//水冷泵测试
R_Test_watercooler_pump(CLK:=Test_watercooler_pump);
IF R_Test_watercooler_pump.Q AND (NOT Motor_work) AND (NOT cooler_motor_Test1)  THEN
    cooler_motor_Test:=TRUE;
	ELSIF R_Test_watercooler_pump.Q AND cooler_motor_Test1 THEN
    cooler_motor_Test:=FALSE;
END_IF
cooler_motor_Test1:=cooler_motor_Test;
//散热风扇测试
R_Test_cooler_fan(CLK:=Test_cooler_fan);
IF R_Test_cooler_fan.Q AND (NOT Motor_work) AND (NOT cooler_fan_Test1)  THEN
    cooler_fan_Test:=TRUE;
    ELSIF R_Test_cooler_fan.Q AND cooler_fan_Test1  THEN
    cooler_fan_Test:=FALSE;
END_IF
cooler_fan_Test1:=cooler_fan_Test;
//扫盘中速测试
R_Test_Sweep_Mspeed(CLK:=Test_Sweep_Mspeed);
IF R_Test_Sweep_Mspeed.Q AND (NOT Sweep_Mspeed_Test1)  THEN
    Sweep_Mspeed_Test:=TRUE;
    Sweep_Lspeed_Test:=FALSE;
ELSIF R_Test_Sweep_Mspeed.Q AND Sweep_Mspeed_Test1  THEN
    Sweep_Mspeed_Test:=FALSE;
END_IF
Sweep_Mspeed_Test1:=Sweep_Mspeed_Test;
//扫盘低速测试
R_Test_Sweep_Lspeed(CLK:=Test_Sweep_Lspeed);
IF R_Test_Sweep_Lspeed.Q AND (NOT Sweep_Lspeed_Test1)  THEN
    Sweep_Lspeed_Test:=TRUE;
    Sweep_Mspeed_Test:=FALSE;
ELSIF R_Test_Sweep_Lspeed.Q AND Sweep_Lspeed_Test1  THEN
    Sweep_Lspeed_Test:=FALSE;
END_IF
Sweep_Lspeed_Test1:=Sweep_Lspeed_Test;
//左扫旋转测试
R_Test_LSweep(CLK:=Test_LSweep);
IF R_Test_LSweep.Q AND (NOT LSweep_Test1)  THEN
    LSweep_Test:=TRUE;
    RSweep_Test:=FALSE;
    ASweep_Test:=FALSE;
ELSIF R_Test_LSweep.Q AND LSweep_Test1  THEN
    LSweep_Test:=FALSE;
END_IF
LSweep_Test1:=LSweep_Test;
//右扫旋转测试
R_Test_RSweep(CLK:=Test_RSweep);
IF R_Test_RSweep.Q AND (NOT RSweep_Test1) THEN
    RSweep_Test:=TRUE;
    LSweep_Test:=FALSE;
    ASweep_Test:=FALSE;
ELSIF R_Test_RSweep.Q AND RSweep_Test1  THEN
    RSweep_Test:=FALSE;
END_IF
RSweep_Test1:=RSweep_Test;
//全扫旋转测试
R_Test_ASweep(CLK:=Test_ASweep);
IF R_Test_ASweep.Q AND (NOT ASweep_Test1) THEN
    RSweep_Test:=FALSE;
    LSweep_Test:=FALSE;
    ASweep_Test:=TRUE;
ELSIF R_Test_ASweep.Q AND ASweep_Test1  THEN
    ASweep_Test:=FALSE;
END_IF
ASweep_Test1 :=ASweep_Test ;
//箱体升降测试
Box_Down_Test:=Test_Box_Down AND (NOT Test_Box_Up) AND (NOT DI_Rod_noDown);
Box_Up_Test:=Test_Box_Up AND (NOT Test_Box_Down);
//吸盘升降测试
Suction_Down_Test:=Test_Suction_Down AND (NOT Test_Suction_Up);
Suction_Up_Test:=Test_Suction_Up AND (NOT Test_Suction_Down);
//箱门开关测试
Boxdoor_close_Test:=Test_Door_Close AND (NOT Test_Door_Open);
Boxdoor_open_Test:=Test_Door_Open AND (NOT Test_Door_Close);
//左扫盘升降测试
LSweep_Up_Test:=Test_LSweep_Up AND (NOT Test_LSweep_Down) AND (NOT DI_Sweep_Down);
LSweep_Down_Test:=Test_LSweep_Down AND (NOT Test_LSweep_Up) AND (NOT DI_Sweep_Up);
//右扫盘升降测试
RSweep_Up_Test:=Test_RSweep_Up AND (NOT Test_RSweep_Down) AND (NOT DI_Sweep_Down);
RSweep_Down_Test:=Test_RSweep_Down AND (NOT Test_RSweep_Up) AND (NOT DI_Sweep_Up);
//左扫盘摆出测试
R_Test_LSweep_out(CLK:=Test_LSweep_out);
IF R_Test_LSweep_out.Q AND (NOT LSweep_out_Test1) THEN
    LSweep_out_Test:=TRUE;
ELSIF R_Test_LSweep_out.Q AND LSweep_out_Test1  THEN
    LSweep_out_Test:=FALSE;
END_IF
LSweep_out_Test1:=LSweep_out_Test;
//右扫盘摆出测试
R_Test_RSweep_out(CLK:=Test_RSweep_out);
IF R_Test_RSweep_out.Q AND (NOT RSweep_out_Test1) THEN
    RSweep_out_Test:=TRUE;
ELSIF R_Test_RSweep_out.Q AND RSweep_out_Test1  THEN
    RSweep_out_Test:=FALSE;
END_IF
RSweep_out_Test1:=RSweep_out_Test;
//左喷杆摆出测试
R_Test_Lrod_OUT(CLK:=Test_Lrod_OUT);
IF R_Test_Lrod_OUT.Q AND (NOT Lrod_OUT_Test1) THEN;
    Lrod_OUT_Test:=TRUE;
ELSIF R_Test_Lrod_OUT.Q AND Lrod_OUT_Test1 THEN;
    Lrod_OUT_Test:=FALSE;
END_IF
Lrod_OUT_Test1:=Lrod_OUT_Test;
//右喷杆摆出测试
R_Test_Rrod_OUT(CLK:=Test_Rrod_OUT);
IF R_Test_Rrod_OUT.Q AND (NOT Rrod_OUT_Test1) THEN;
    Rrod_OUT_Test:=TRUE;
ELSIF R_Test_Rrod_OUT.Q AND Rrod_OUT_Test1 THEN;
    Rrod_OUT_Test:=FALSE;
END_IF
Rrod_OUT_Test1 :=Rrod_OUT_Test;
//左喷杆喷水测试
R_Test_Lrod_water(CLK:=Test_Lrod_water);
IF R_Test_Lrod_water.Q AND (NOT Lrod_water_Test1) THEN
    Lrod_water_Test:=TRUE;
ELSIF R_Test_Lrod_water.Q AND Lrod_water_Test1 THEN
    Lrod_water_Test:=FALSE;
END_IF
Lrod_water_Test1:=Lrod_water_Test;
//右喷杆喷水测试
R_Test_Rrod_water(CLK:=Test_Rrod_water);
IF R_Test_Rrod_water.Q AND (NOT Rrod_water_Test1) THEN
    Rrod_water_Test:=TRUE;
ELSIF R_Test_Rrod_water.Q AND Rrod_water_Test1 THEN
    Rrod_water_Test:=FALSE;
END_IF
Rrod_water_Test1:=Rrod_water_Test;
//吸嘴喷杆喷水测试
R_Test_Suction_water(CLK:=Test_Suction_water);
IF R_Test_Suction_water.Q AND (NOT Suction_water_Test1) THEN
    Suction_water_Test:=TRUE;
ELSIF R_Test_Suction_water.Q AND Suction_water_Test1 THEN
    Suction_water_Test:=FALSE;
END_IF
Suction_water_Test1:=Suction_water_Test;
//高压冲洗测试
R_Test_Hpre_wash(CLK:=Test_Hpre_wash);
IF R_Test_Hpre_wash.Q AND (NOT Hpre_wash_Test1) THEN
    Hpre_wash_Test:=TRUE;
ELSIF R_Test_Hpre_wash.Q AND Hpre_wash_Test1 THEN
    Hpre_wash_Test:=FALSE;
END_IF
Hpre_wash_Test1:=Hpre_wash_Test;
//自洁测试
R_Test_selfclean(CLK:=Test_selfclean);
IF R_Test_selfclean.Q AND (NOT selfclean_water_Test1) THEN
    selfclean_water_Test:=TRUE;
END_IF
IF R_Test_selfclean.Q AND selfclean_water_Test1 THEN
    selfclean_water_Test:=FALSE;
END_IF
selfclean_water_Test1 :=selfclean_water_Test;
//高压水泵啮合测试
R_Test_Hpre_pump_gearin(CLK:=Test_Hpre_pump_gearin);
IF R_Test_Hpre_pump_gearin.Q AND (NOT Hpress_pump_gearin_Test1) THEN
    Hpress_pump_gearin_Test:=TRUE;
ELSIF (R_Test_Hpre_pump_gearin.Q AND Hpress_pump_gearin_Test1) OR T_pumpClutch.Q THEN
    Hpress_pump_gearin_Test:=FALSE;
END_IF
Hpress_pump_gearin_Test1 :=Hpress_pump_gearin_Test;
(*发动机工作时，水箱缺水时，延时10S高压水泵分离 *)
T_pumpClutch(IN:=Motor_work AND DI_cleanwater_LOW_ALM  AND Hpress_pump_gearin_Test ,PT:=T#10S);
//喷雾降尘泵测试
R_Test_fogpump(CLK:=Test_fogpump);
IF R_Test_fogpump.Q AND (NOT Fog_pump_Test1) THEN
    Fog_pump_Test:=TRUE;
ELSIF (R_Test_fogpump.Q AND Fog_pump_Test1) OR T_Fog_pump_Test.Q THEN
    Fog_pump_Test:=FALSE;
END_IF
Fog_pump_Test1 :=Fog_pump_Test;
(*发动机工作时，水箱缺水时，延时90S隔膜泵停止 *)
T_Fog_pump_Test(IN:=DI_cleanwater_LOW_ALM  AND Fog_pump_Test ,PT:=T#90S);
//污水泵测试
R_Test_wastewater_pump(CLK:=Test_wastewater_pump);
IF R_Test_wastewater_pump.Q AND (NOT Wastewater_pump_Test1) THEN
    Wastewater_pump_Test:=TRUE;
ELSIF R_Test_wastewater_pump.Q AND Wastewater_pump_Test1 THEN
    Wastewater_pump_Test:=FALSE;
END_IF
Wastewater_pump_Test1 :=Wastewater_pump_Test;
//污水泵球阀测试
R_Test_wastewater_valve(CLK:=Test_wastewater_valve);
IF R_Test_wastewater_valve.Q AND (NOT Wastewater_valve_Test1) THEN
    Wastewater_valve_Test:=TRUE;
ELSIF R_Test_wastewater_valve.Q AND Wastewater_valve_Test1 THEN
    Wastewater_valve_Test:=FALSE;
END_IF
Wastewater_valve_Test1 :=Wastewater_valve_Test;
//备用动力测试
R_Test_backup_power(CLK:=Test_backup_power);
IF R_Test_backup_power.Q AND (NOT Backup_power_Test1) THEN
    Backup_power_Test:=TRUE;
ELSIF (R_Test_backup_power.Q AND Backup_power_Test1) OR T_Backup_power_Test.Q THEN
    Backup_power_Test:=FALSE;
END_IF
Backup_power_Test1 :=Backup_power_Test;
(*备用动力打开90S后自动关闭 *)
T_Backup_power_Test(IN:=Backup_power_Test ,PT:=T#90S);
Backup_power_Test_warn:=Backup_power_Test AND (NOT DI_backup_power_open);

//点喷测试
Test_pointshoot_up := Pointshoot_up_Test AND NOT Pointshoot_down_Test;
Test_pointshoot_down := Pointshoot_down_Test AND NOT Pointshoot_up_Test; 
Test_pointshoot_left := Pointshoot_left_Test AND NOT Pointshoot_right_Test; 
Test_pointshoot_right := Pointshoot_right_Test AND NOT Pointshoot_left_Test;

END_PROGRAM

// Changsha_Xiangji_ARM_Cortex_A9_xilinx_zynq7000_linux/Application/CAN_COMM/prg_can0
PROGRAM prg_can0   //CAN0   与底盘和显示屏通信
VAR
	hCan0:CAA.HANDLE:=0;
    CanWriteData : ARRAY[0..7] OF BYTE;
    CanWriteMsgID:UDINT;
	CanReadData : ARRAY[0..7] OF BYTE;  
	CanReadMsgID:UDINT;
	bModifyTimeFlag :BOOL := FALSE;
	
	//通过CAN总线从底盘读到的信息
	can_data_ready:BOOL := FALSE;
	can_data_speed:BYTE := 0;
	can_data_soc:BYTE := 0;
	
	//通过CAN总线从显示屏读到的信息
	c00byte0bit0_both_wash_sweep:BOOL := FALSE;
	c00byte0bit1_left_wash_sweep:BOOL := FALSE;
	c00byte0bit2_right_wash_sweep:BOOL := FALSE;
	c00byte0bit3_both_sweep:BOOL := FALSE;
	c00byte0bit4_left_sweep:BOOL := FALSE;
	c00byte0bit5_right_sweep:BOOL := FALSE;
	c00byte0bit6_both_wash:BOOL := FALSE;
	c00byte0bit7_left_wash:BOOL := FALSE;
	
	c00byte1bit0_right_wash:BOOL := FALSE;
	c00byte1bit1_stop_sweep:BOOL := FALSE;
	c00byte1bit2_start_motor:BOOL := FALSE;
	c00byte1bit3_stop_motor:BOOL := FALSE;
	c00byte1bit4_speed_add:BOOL := FALSE;
	c00byte1bit5_speed_dec:BOOL := FALSE;
	c00byte1bit6_normal_speed:BOOL := FALSE;
	c00byte1bit7_high_speed:BOOL := FALSE;
	
	c00byte2bit0_garbage_close:BOOL := FALSE;
	c00byte2bit1_garbage_open:BOOL := FALSE;
	c00byte2bit2_garbage_up:BOOL := FALSE;
	c00byte2bit3_garbage_down:BOOL := FALSE;
	c00byte2bit4_fog_bump:BOOL := FALSE;
	c00byte2bit5_selfclean:BOOL := FALSE;
	c00byte2bit6_wastewater_pump:BOOL := FALSE;
	c00byte2bit7_res :BOOL := FALSE;
	
	c00byte3bit0_sweep_high:BOOL := FALSE;
	c00byte3bit1_sweep_middle:BOOL := FALSE;
	c00byte3bit2_sweep_low:BOOL := FALSE;
	c00byte3bit3_highpress_wash:BOOL := FALSE;
	c00byte3bit4_pointshoot_up:BOOL := FALSE;
	c00byte3bit5_pointshoot_down:BOOL := FALSE;
	c00byte3bit6_pointshoot_left:BOOL := FALSE;
	c00byte3bit7_pointshoot_right:BOOL := FALSE;

	c00byte4bit0_drain_start:BOOL := FALSE;
	c00byte4bit1_drain_auto:BOOL := FALSE;
	c00byte4bit2_drain_manual:BOOL := FALSE;
	c00byte4bit3_left_drain:BOOL := FALSE;
	c00byte4bit4_right_drain:BOOL := FALSE;
	c00byte4bit5_sub_drain:BOOL := FALSE;
	c00byte4bit6_selfclean_drain:BOOL := FALSE;
	c00byte4bit7_spout_drain:BOOL := FALSE;
	
	c00byte6bit0_func_test:BOOL := FALSE;
	c00byte6bit1_change_sweeper:BOOL := FALSE;
	c00byte6bit2_intelligent:BOOL := FALSE;
	c00byte6bit3_cleanly:BOOL := FALSE;
	c00byte6bit4_normal:BOOL := FALSE;
	c00byte6bit5_dirty:BOOL := FALSE;
	
	c01byte0bit3_test_watercooler_pump:BOOL := FALSE;
	c01byte0bit4_test_cooler_fan:BOOL := FALSE;
	
	c01byte1bit0_test_sweeper_middle:BOOL := FALSE;
	c01byte1bit1_test_sweeper_low:BOOL := FALSE;
	c01byte1bit2_test_left_sweeper:BOOL := FALSE;
	c01byte1bit3_test_right_sweeper:BOOL := FALSE;
	c01byte1bit4_test_both_sweeper:BOOL := FALSE;
	c01byte1bit5_test_box_down:BOOL := FALSE;
	c01byte1bit6_test_box_up:BOOL := FALSE;
	c01byte1bit7_test_sucker_down:BOOL := FALSE;
	
	c01byte2bit0_test_sucker_up:BOOL := FALSE;
	c01byte2bit1_test_box_open:BOOL := FALSE;
	c01byte2bit2_test_box_close:BOOL := FALSE;
	
	c01byte2bit6_test_left_sweeper_down:BOOL := FALSE;
	c01byte2bit7_test_left_sweeper_up:BOOL := FALSE;
	
	c01byte3bit0_test_right_sweeper_down:BOOL := FALSE;
	c01byte3bit1_test_right_sweeper_up:BOOL := FALSE;
	c01byte3bit2_test_left_sweeper_out:BOOL := FALSE;
	c01byte3bit3_test_right_sweeper_out:BOOL := FALSE;
	c01byte3bit4_test_left_shooter_out:BOOL := FALSE;
	c01byte3bit5_test_right_shooter_out:BOOL := FALSE;
	c01byte3bit6_test_left_shooter_water:BOOL := FALSE;
	c01byte3bit7_test_right_shooter_water:BOOL := FALSE;
	
	c01byte4bit0_test_sucker_water:BOOL := FALSE;
	c01byte4bit1_test_highpress_wash:BOOL := FALSE;
	c01byte4bit2_test_selfclean:BOOL := FALSE;
	c01byte4bit3_test_highpress_pump_gearin:BOOL := FALSE;
	c01byte4bit4_test_fogpump:BOOL := FALSE;
	c01byte4bit5_test_pointshoot_up:BOOL := FALSE;
    c01byte4bit6_test_pointshoot_down:BOOL := FALSE;
    c01byte4bit7_test_pointshoot_left:BOOL := FALSE;
	
	c01byte5bit0_test_pointshoot_right:BOOL := FALSE;
	c01byte5bit2_test_wastewater_pump:BOOL := FALSE;
	c01byte5bit3_test_wastewater_valve:BOOL := FALSE;
	
	c01byte6bit0_test_backup_power:BOOL := FALSE;
	
	c02byte45_speed_change :UINT := 0;
	c02byte67_sub_motor_min_speed:UINT := 0;
	
	c03byte01_normal_speed:UINT := 0;
	c03byte23_high_speed:UINT := 0;
	c03byte45_sweeper_speed:UINT := 0;
	
	c04byte01_highpress_pump_overspeed_warning:UINT := 0;
	c04byte23_highpress_pump_overspeed_stop:UINT := 0;
	c04byte45_sub_motor_max_speed:UINT := 0;
	c04byte67_sub_motor_idle_speed:UINT := 0;
	
	c05byte01_clean_low_speed:UINT := 0;
    c05byte23_clean_midlow_speed:UINT := 0;
    c05byte45_clean_midhigh_speed:UINT := 0;
    c05byte67_clean_high_speed:UINT := 0;
	
	c06byte01_normal_low_speed:UINT := 0;
    c06byte23_normal_midlow_speed:UINT := 0;
    c06byte45_normal_midhigh_speed:UINT := 0;
    c06byte67_normal_high_speed:UINT := 0;
	
	c07byte01_dirty_low_speed:UINT := 0;
    c07byte23_dirty_midlow_speed:UINT := 0;
    c07byte45_dirty_midhigh_speed:UINT := 0;
    c07byte67_dirty_high_speed:UINT := 0;
	
	//通过CAN总线发送到显示屏的信息
	s00byte0bit0_res:BOOL := FALSE;
	
	s00byte1bit0_res:BOOL := FALSE;
	s00byte1bit1_wastewater_full:BOOL := FALSE;
	s00byte1bit2_oil_filter_block:BOOL := FALSE;
	s00byte1bit3_oil_low:BOOL := FALSE;
	s00byte1bit4_res:BOOL := FALSE;
	s00byte1bit5_tank_no_water:BOOL := FALSE;
	s00byte1bit6_res:BOOL := FALSE;
	s00byte1bit7_back_error_stop:BOOL := FALSE;
	
	s00byte2bit0_wastewater_full_stop:BOOL := FALSE;
	s00byte2bit1_electronic_power_fault:BOOL := FALSE;
	s00byte2bit2_highpress_pump_overspeed_warning:BOOL := FALSE;
	s00byte2bit3_highpress_pump_overspeed_stop:BOOL := FALSE;
	s00byte2bit4_please_close_test:BOOL := FALSE;
	s00byte2bit5_being_back:BOOL := FALSE;
	s00byte2bit6_please_open_motor:BOOL := FALSE;
	s00byte2bit7_please_open_test:BOOL := FALSE;
	
	s00byte3bit0_air_press_low:BOOL := FALSE;
	s00byte3bit1_back_the_truck:BOOL := FALSE;
	s00byte3bit2_res:BOOL := FALSE;
	s00byte3bit3_highpress_pump_not_gearin:BOOL := FALSE;
	s00byte3bit4_water_valve_not_on:BOOL := FALSE;
	s00byte3bit5_highpress_blow_valve_not_on:BOOL := FALSE;
	s00byte3bit6_highpress_water_valve_not_on:BOOL := FALSE;
	s00byte3bit7_please_open_box_door:BOOL := FALSE;
	
	s00byte4bit0_pump_valve_not_no:BOOL := FALSE;
	s00byte4bit1_pump_press_fault:BOOL := FALSE;
	s00byte4bit2_fault_stop:BOOL := FALSE;
	s00byte4bit3_please_putdown_supporter:BOOL := FALSE;
	
	s00byte4bit6_chassis_can_fault:BOOL := FALSE;
	s00byte4bit7_motordriver_can_fault:BOOL :=FALSE;
	
	s00byte5bit0_sub_wastebox_error:BOOL := FALSE;
	s00byte5bit1_sub1_wastebox_full:BOOL := FALSE;
	s00byte5bit2_sub2_wastebox_full:BOOL := FALSE;
	s00byte5bit3_water_release_valve_not_close:BOOL := FALSE;
	s00byte5bit4_water_release_valve_not_copen:BOOL := FALSE;
	s00byte5bit5_backup_power_on:BOOL := FALSE;
	s00byte5bit6_power_low_20percent:BOOL := FALSE;
	s00byte5bit7_chassis_no_high_voltage:BOOL := FALSE;
	
	s00byte6bit0_cleanwater_LOW:BOOL := FALSE;
	s00byte6bit1_highpress_water_valve_on:BOOL := FALSE;
	s00byte6bit2_box_door_close:BOOL := FALSE;
	s00byte6bit3_highpress_blow_valve_on:BOOL := FALSE;
	s00byte6bit4_air_press_low:BOOL := FALSE;
	s00byte6bit5_wastewater_full:BOOL := FALSE;
	s00byte6bit6_supporter_nodown:BOOL := FALSE;
	s00byte6bit7_backup_power_open:BOOL := FALSE;
	
	s00byte7bit0_water_release_valve:BOOL := FALSE;
	s00byte7bit4_fog_pump_press_ok:BOOL := FALSE;
	s00byte7bit5_oil_level_low:BOOL := FALSE;
	s00byte7bit6_oil_filter_block:BOOL := FALSE;
	
	s01byte0bit0_power_on:BOOL := FALSE;
	s01byte0bit1_back_the_truck:BOOL := FALSE;
	s01byte0bit2_oil_release_valve:BOOL := FALSE;
	s01byte0bit3_cleanwater_low:BOOL := FALSE;
	s01byte0bit4_auxiliary1_warte_H:BOOL := FALSE;
	s01byte0bit5_auxiliary2_warte_H:BOOL := FALSE;
	s01byte0bit6_sweeper_up:BOOL := FALSE;
    s01byte0bit7_sweeper_down:BOOL := FALSE;
	
	s01byte1bit0_sweeper_out:BOOL := FALSE;
	s01byte1bit1_sweeper_return:BOOL := FALSE;
	
	s01byte3bit0_left_sweeper_down:BOOL := FALSE;
    s01byte3bit1_left_sweeper_up:BOOL := FALSE;
    s01byte3bit2_right_sweeper_down:BOOL := FALSE;
    s01byte3bit3_right_sweeper_up:BOOL := FALSE;
    s01byte3bit4_left_sweeper_out:BOOL := FALSE;
    s01byte3bit5_right_sweeper_out:BOOL := FALSE;
    s01byte3bit6_left_shooter_out:BOOL := FALSE;
    s01byte3bit7_right_shooter_out:BOOL := FALSE;

    s01byte4bit5_water_release_valve_open:BOOL := FALSE;
    s01byte4bit6_left_shooter_open:BOOL := FALSE;
    s01byte4bit7_right_shooter_open:BOOL := FALSE;
	
//	s01byte4bit4_oil_release_valve:BOOL := FALSE;
//	s01byte4bit5_sweeper_middle_speed:BOOL := FALSE;
//	s01byte4bit6_sweeper_low_speed:BOOL := FALSE;
//	s01byte4bit7_left_sweeper_back:BOOL := FALSE;
	
    s01byte5bit0_sucker_shooter_water:BOOL := FALSE;
    s01byte5bit1_fog_pump_open:BOOL := FALSE;
    s01byte5bit2_selfclean_shooter_water:BOOL := FALSE;
    s01byte5bit3_high_sub_shooter_water:BOOL := FALSE;
    s01byte5bit4_Spump_open:BOOL := FALSE;
    s01byte5bit5_engine_en:BOOL := FALSE;
    s01byte5bit6_watercooler_pump_open:BOOL := FALSE;
    s01byte5bit7_cooler_fan_open:BOOL := FALSE;
	
    s01byte6bit0_backup_power_open:BOOL := FALSE;
    s01byte6bit1wastewater_valve_open:BOOL := FALSE;
    s01byte6bit2_wastewater_pump_open:BOOL := FALSE;
    s01byte6bit3_oil_release_valve_open:BOOL := FALSE;
    s01byte6bit4_sweep_middle_open:BOOL := FALSE;
    s01byte6bit5_sweep_low_open:BOOL := FALSE;
    s01byte6bit6_right_sweep_open:BOOL := FALSE;
    s01byte6bit7_left_both_sweep_open:BOOL := FALSE;
	
    s01byte7bit0_right_both_sweep_open:BOOL := FALSE;
    s01byte7bit1_box_down:BOOL := FALSE;
    s01byte7bit2_box_up:BOOL := FALSE;
    s01byte7bit3_sucker_down:BOOL := FALSE;
    s01byte7bit4_sucker_up:BOOL := FALSE;
    s01byte7bit5_box_open:BOOL := FALSE;
    s01byte7bit6_box_close:BOOL := FALSE;
	
	s02byte0bit67_right_shooter_out:BYTE := 0;
	
	s02byte1bit01_left_shooter_out:BYTE := 0;
	s02byte1bit23_waterpump_gearin:BYTE := 0;
	s02byte1bit45_left_shooter_valve_open:BYTE := 0;
	s02byte1bit67_right_shooter_valve_open:BYTE := 0;
	
	s02byte2bit01_sucker_shooter_valve_open:BYTE := 0;
	s02byte2bit23_selfclean_shooter_valve_open:BYTE := 0;
	s02byte2bit45_high_sub_shooter_valve_open:BYTE := 0;
	s02byte2bit67_water_release_valve:BYTE := 0;
	
	s02byte3bit01_oil_release_valve:BYTE := 0;
	s02byte3bit23_sweeper_middle_speed:BYTE := 0;
	s02byte3bit45_sweeper_low_speed:BYTE := 0;
	s02byte3bit67_left_sweeper_back:BYTE := 0;
	
	s02byte4bit01_left_sweeper_down:BYTE := 0;
	s02byte4bit23_right_sweeper_back:BYTE := 0;
	s02byte4bit45_right_sweeper_down:BYTE := 0;
	s02byte4bit67_left_all_sweep:BYTE := 0;
	
	s02byte5bit01_right_sweep:BYTE := 0;
	s02byte5bit23_res:BYTE := 0;
	
	s02byte6bit01_right_all_sweep:BYTE := 0;
	s02byte6bit23_box_down:BYTE := 0;
	s02byte6bit45_box_up:BYTE := 0;
	s02byte6bit67_sucker_up:BYTE := 0;
	
	s02byte7bit01_sucker_down:BYTE := 0;
	s02byte7bit23_boxdoor_close:BYTE := 0;
	s02byte7bit45_boxdoor_open:BYTE := 0;
	s02byte7bit67_cleanwater_pump:BYTE := 0;
	
	s03byte0bit01_res:BYTE := 0;
	s03byte0bit23_water_coller_motor:BYTE := 0;
	s03byte0bit45_cooler_fan:BYTE := 0;
	s03byte0bit67_lowpress_pump:BYTE := 0;
	
	s03byte3bit0_all_wash_sweep:BOOL := FALSE;
	s03byte3bit1_left_wash_sweep:BOOL := FALSE;
	s03byte3bit2_right_wash_sweep:BOOL := FALSE;
	s03byte3bit3_all_sweep:BOOL := FALSE;
	s03byte3bit4_left_sweep:BOOL := FALSE;
	s03byte3bit5_right_sweep:BOOL := FALSE;
	s03byte3bit6_all_wash:BOOL := FALSE;
	s03byte3bit7_left_wash:BOOL := FALSE;
	
	s03byte4bit0_right_wash:BOOL := FALSE;
	s03byte4bit1_stop_sweep:BOOL := FALSE;
	s03byte4bit2_fog_pump:BOOL := FALSE;
	s03byte4bit3_selfclean:BOOL := FALSE;
	s03byte4bit4_boxdoor_close:BOOL := FALSE;
	s03byte4bit5_boxdoor_open:BOOL := FALSE;
	s03byte4bit6_box_up:BOOL := FALSE;
	s03byte4bit7_box_down:BOOL := FALSE;
	
	s03byte5bit0_motor_start:BOOL := FALSE;
	s03byte5bit1_motor_stop:BOOL := FALSE;
	s03byte5bit4_normal_speed:BOOL := FALSE;
	s03byte5bit5_high_speed:BOOL := FALSE;
	s03byte5bit6_sweeper_high_speed:BOOL := FALSE;
	s03byte5bit7_sweeper_middle_spped:BOOL := FALSE;
	
	s03byte6bit0_sweeper_low_speed:BOOL := FALSE;
	s03byte6bit1_highpress_wash:BOOL := FALSE;
	s03byte6bit2_drain_start:BOOL := FALSE;
	s03byte6bit3_drain_auto:BOOL := FALSE;
	s03byte6bit4_drain_manual:BOOL := FALSE;
	s03byte6bit5_drain_left_shooter:BOOL := FALSE;
	s03byte6bit6_drain_right_shooter:BOOL := FALSE;
	s03byte6bit7_sub_drain:BOOL := FALSE;
	
	s03byte7bit0_drain_selfclean:BOOL := FALSE;
	s03byte7bit1_change_sweeper:BOOL := FALSE;
	s03byte7bit2_func_test:BOOL := FALSE;
	s03byte7bit3_intelligent:BOOL := FALSE;
	s03byte7bit4_cleanly:BOOL := FALSE;
	s03byte7bit5_normal:BOOL := FALSE;
	s03byte7bit6_dirty:BOOL := FALSE;
	s03byte7bit7_wastewater_pump:BOOL := FALSE;
	
	s04byte0bit0_point_shoot_up:BOOL := FALSE;
	s04byte0bit1_point_shoot_down:BOOL := FALSE;
	s04byte0bit2_point_shoot_left:BOOL := FALSE;
	s04byte0bit3_point_shoot_right:BOOL := FALSE;
	s04byte0bit4_sucker_shooter_drain:BOOL := FALSE;
	
	s04byte1bit3_test_cooler_motor:BOOL := FALSE;
	s04byte1bit4_test_cooler_fan:BOOL := FALSE;
	s04byte1bit5_test_sweeper_middle:BOOL := FALSE;
	s04byte1bit6_test_sweeper_low:BOOL := FALSE;
	s04byte1bit7_test_left_sweep:BOOL := FALSE;
	
	s04byte2bit0_test_right_sweep:BOOL := FALSE;
	s04byte2bit1_test_all_sweep:BOOL := FALSE;
	s04byte2bit2_test_box_down:BOOL := FALSE;
	s04byte2bit3_test_box_up:BOOL := FALSE;
	s04byte2bit4_test_sucker_down:BOOL := FALSE;
	s04byte2bit5_test_sucker_up:BOOL := FALSE;
	s04byte2bit6_test_boxdoor_open:BOOL := FALSE;
	s04byte2bit7_test_boxdoor_close:BOOL := FALSE;
	
	s04byte3bit0_test_left_sweeper_down:BOOL := FALSE;
	s04byte3bit1_test_left_sweeper_up:BOOL := FALSE;
	s04byte3bit2_test_right_sweeper_down:BOOL := FALSE;
	s04byte3bit3_test_right_sweeper_up:BOOL := FALSE;
	s04byte3bit4_test_left_shooter_out:BOOL := FALSE;
	s04byte3bit5_test_right_shooter_out:BOOL := FALSE;
	s04byte3bit6_test_left_shooter_water:BOOL := FALSE;
	s04byte3bit7_test_right_shooter_water:BOOL := FALSE;
	
	s04byte4bit0_test_sucker_water:BOOL := FALSE;
	s04byte4bit1_test_highpress_wash:BOOL := FALSE;
	s04byte4bit2_test_selfclean:BOOL := FALSE;
	s04byte4bit3_test_highpress_pump_gearin:BOOL := FALSE;
	s04byte4bit4_test_fog_pump:BOOL := FALSE;
	s04byte4bit5_test_left_sweeper_out:BOOL := FALSE;
	s04byte4bit6_test_right_sweeper_out:BOOL := FALSE;
	s04byte4bit7_test_wastewater_pump:BOOL := FALSE;
	
	s04byte5bit0_test_wastewater_valve:BOOL := FALSE;
	s04byte5bit1_test_backup_power:BOOL := FALSE;
	s04byte5bit6_motor_starting:BOOL := FALSE;
	s04byte5bit7_system_running:BOOL := FALSE;
	
	s05byte45_speed_change_value:UINT := 0;
	s05byte67_sub_motor_min_speed:UINT := 0;
	
	s06byte01_normal_speed:UINT := 0;
	s06byte23_high_speed:UINT := 0;
	s06byte45_sweeper_speed:UINT := 0;
	
	s07byte01_highpress_pump_high_speed:UINT := 0;
	s07byte23_highpress_pump_high_speed_stop:UINT := 0;
	s07byte45_sub_motor_max_speed:UINT := 0;
	s07byte67_sub_motor_idle_speed:UINT := 0;
	
	s08byte01_real_torque:UINT := 0;
	s08byte23_real_speed:UINT := 0;
	s08byte45_bus_voltage:UINT := 0;
	s08byte67_phase_current:UINT := 0;
	
	s09byte01_max_dirve_torque:UINT := 0;
	s09byte23_max_brake_torque:UINT := 0;
	s09byte4_temp_controller:BYTE := 0;
	s09byte5_temp_motor:BYTE := 0;
	s09byte67_motor_max_speed:UINT := 0;
	
	s10byte0bit23_direction_cw:BYTE := 0;
	s10byte0bit45_motor_mode:BYTE := 0;
	s10byte0bit67_motor_stat:BYTE := 0;
	
	s10byte1bit01_bus_low_voltage:BYTE := 0;
	s10byte1bit23_bus_high_voltage:BYTE := 0;
	s10byte1bit45_ctrller_high_temp:BYTE := 0;
	s10byte1bit67_motor_high_temp:BYTE := 0;
	
	s10byte2bit01_igbt_fault:BYTE := 0;
	s10byte2bit23_overspeed:BYTE := 0;
	s10byte2bit45_comm_error:BYTE := 0;
	s10byte2bit67_short:BYTE := 0;
	
	s10byte3bit01_motor_overload:BYTE := 0;
	s10byte3bit23_selfcheck_fault:BYTE := 0;
	s10byte3bit45_low_voltage:BYTE := 0;
	s10byte3bit67_sensor_fault:BYTE := 0;
	
	s11byte0_chassis_power_percent:BYTE := 0;
	s11byte1_res :BYTE := 0;
	s11byte23_speed_set_value:UINT := 0;
	s11byte45_version:UINT := 0;
	
    //电机
	
	hReceiver1:CAA.HANDLE;
	hReceiver2:CAA.HANDLE;
	hReceiver3:CAA.HANDLE;
	
	//显示屏 0x0c00 074f ~ 0x0c07 074f
	hRecver_screen:CAA.HANDLE;
	
	tmp_byte:BYTE;
	tmp_uint:UINT;
	Err:CAA.ERROR;
	
	hMsg : CAA.HANDLE;
	nReceived : CAA.COUNT;
	nAvailable: CAA.COUNT;
	ReadErr   : CAA.ERROR;
	MsgID     : CL2I.COBID;	
	pRxData :POINTER TO CL2I.DATA;
	//电机CAN通信标志位
	nReceived1 : CAA.COUNT;
	
	can_stat : DINT := 0;
	
	n: INT := 0;
	m: INT := 0;
END_VAR

CASE can_stat OF
	0:   //init can port0 and port1
		hCan0 := cl2.DriverOpenH(usiNetId:=0,uiBaudRate:=250,xSupport29Bits:=TRUE,ctMessages:=100,peError:=ADR(Err));	 //CAN1
		IF hCan0 > 0 THEN
			can_stat := 10;
		END_IF
	
	10: //create receiver for data
		//接收驱动器信息1: ID:0x0C112AEE,  
	  	hReceiver1 := CL2.CreateMaskReceiver(hDriver := hCan0,
			cobIdValue := 16#0C112AEE, //cobID value
			cobIdMask := 16#FFFFFFFF, //cobID mask ==> all bits of value are relevant									
			xRTRValue := FALSE, //no RTR messages
			xRTRMask := FALSE, //activate RTR filter ==> xRTRValue will be checked
			x29BitIdValue := TRUE, //29 bit CAN messages
			x29BitIdMask := TRUE, //activate 29 bit filter ==> x29BitIdValue will be checked
			xTransmitValue := FALSE, //only receive messages, no transmit message loopback
			xTransmitMask := FALSE, //activate transmit mask filter ==> xTransmitValue will be checked
			xAlwaysNewest := FALSE, //FALSE := receiver with queue; TRUE: only newest message
			eEvent := CB.EVENT.NO_EVENT,  //no receive event
			xEnableSyncWindow := FALSE, //not implemented
			peError := ADR(Err) //optional pointer to error
			);
		//接收驱动器信息2: ID:0x0C122AEE	
	  	hReceiver2 := CL2.CreateMaskReceiver(hDriver := hCan0,
			cobIdValue := 16#0C122AEE, //cobID value
			cobIdMask := 16#FFFFFFFF, //cobID mask ==> all bits of value are relevant									
			xRTRValue := FALSE, //no RTR messages
			xRTRMask := FALSE, //activate RTR filter ==> xRTRValue will be checked
			x29BitIdValue := TRUE, //29 bit CAN messages
			x29BitIdMask := TRUE, //activate 29 bit filter ==> x29BitIdValue will be checked
			xTransmitValue := FALSE, //only receive messages, no transmit message loopback
			xTransmitMask := FALSE, //activate transmit mask filter ==> xTransmitValue will be checked
			xAlwaysNewest := FALSE, //FALSE := receiver with queue; TRUE: only newest message
			eEvent := CB.EVENT.NO_EVENT, //no receive event
			xEnableSyncWindow := FALSE, //not implemented
			peError := ADR(Err) //optional pointer to error
			);	
		
		//接收驱动器信息3: ID:0x0C132AEE
		hReceiver3 := CL2.CreateMaskReceiver(hDriver := hCan0,
			cobIdValue := 16#0C132AEE, //cobID value
			cobIdMask := 16#FFFFFFFF, //cobID mask ==> all bits of value are relevant									
			xRTRValue := FALSE, //no RTR messages
			xRTRMask := FALSE, //activate RTR filter ==> xRTRValue will be checked
			x29BitIdValue := TRUE, //no 29 bit CAN messages
			x29BitIdMask := TRUE, //activate 29 bit filter ==> x29BitIdValue will be checked
			xTransmitValue := FALSE, //only receive messages, no transmit message loopback
			xTransmitMask := FALSE, //activate transmit mask filter ==> xTransmitValue will be checked
			xAlwaysNewest := FALSE, //FALSE := receiver with queue; TRUE: only newest message
			eEvent := CB.EVENT.NO_EVENT, //no receive event
			xEnableSyncWindow := FALSE, //not implemented
			peError := ADR(Err) //optional pointer to error
		);
				//创建接收显示屏信息的接收器: ID:0x0cxx074f
		hRecver_screen := CL2.CreateMaskReceiver(hDriver := hCan0,
			cobIdValue := 16#0C00074F, //cobID value  
			cobIdMask := 16#FFF8FFFF, //cobID mask	0c00074f,0c01074f,0c02074f,0c03074f,							
			xRTRValue := FALSE, //no RTR messages
			xRTRMask := FALSE, //activate RTR filter ==> xRTRValue will be checked
			x29BitIdValue := TRUE, //no 29 bit CAN messages
			x29BitIdMask := TRUE, //activate 29 bit filter ==> x29BitIdValue will be checked
			xTransmitValue := FALSE, //only receive messages, no transmit message loopback
			xTransmitMask := FALSE, //activate transmit mask filter ==> xTransmitValue will be checked
			xAlwaysNewest := FALSE, //FALSE := receiver with queue; TRUE: only newest message
			eEvent := CB.EVENT.NO_EVENT, //no receive event
			xEnableSyncWindow := FALSE, //not implemented
			peError := ADR(Err) //optional pointer to error
		);
		
		IF (hReceiver1 <> 0 AND hReceiver2 <> 0 AND hReceiver3 <> 0 AND hRecver_screen <> 0) THEN
			 can_stat := 20;
		ELSE
			RETURN;
		END_IF
	20:  //receive data
		//接收驱动器信息1: ID:0x0C112AEE,  
		nReceived1 := cl2.GetMsgCount(hReceiverId :=hReceiver1, peError := ADR(ReadErr));
		m:=m+1;
		WHILE nReceived1 > 0 DO
			m:=0;
			hMsg := cl2.Read(hReceiverId :=hReceiver1,pctMsgLeft:=ADR(nAvailable),peError:=ADR(ReadErr));
			pRxData := cl2.GetMessageDataPointer(hMessage:= hMsg,peError:=ADR(ReadErr));	
			get_buf_0C112AEE(pRxData);
			cl2.FreeMessage(hMsg);
	        nReceived1 := cl2.GetMsgCount(hReceiverId :=hReceiver1, peError := ADR(ReadErr));
		END_WHILE


		//接收驱动器信息2: ID:0x0C122AEE
		nReceived1 := cl2.GetMsgCount(hReceiverId :=hReceiver2, peError := ADR(ReadErr));
		WHILE nReceived1 > 0 DO
			hMsg := cl2.Read(hReceiverId :=hReceiver2,pctMsgLeft:=ADR(nAvailable),peError:=ADR(ReadErr));
			pRxData := cl2.GetMessageDataPointer(hMessage:= hMsg,peError:=ADR(ReadErr));	
			get_buf_0C122AEE(pRxData);
			cl2.FreeMessage(hMsg);
			nReceived1 := cl2.GetMsgCount(hReceiverId :=hReceiver2, peError := ADR(ReadErr));
		END_WHILE

		//接收驱动器信息3: ID:0x0C132AEE
		nReceived1 := cl2.GetMsgCount(hReceiverId :=hReceiver3, peError := ADR(ReadErr));
		WHILE nReceived1 > 0 DO
			hMsg := cl2.Read(hReceiverId :=hReceiver3,pctMsgLeft:=ADR(nAvailable),peError:=ADR(ReadErr));
			pRxData := cl2.GetMessageDataPointer(hMessage:= hMsg,peError:=ADR(ReadErr));	
			get_buf_0C132AEE(pRxData);
			cl2.FreeMessage(hMsg);	
			nReceived1 := cl2.GetMsgCount(hReceiverId :=hReceiver3, peError := ADR(ReadErr));
		END_WHILE
        
		
       //接收显示屏信息: ID:0x0cXX074f
		nReceived := cl2.GetMsgCount(hReceiverId :=hRecver_screen, peError := ADR(ReadErr));
		n:=n+1;
		WHILE nReceived > 0 DO
			n:=0;
			hMsg := cl2.Read(hReceiverId :=hRecver_screen,pctMsgLeft:=ADR(nAvailable),peError:=ADR(ReadErr));
			pRxData := cl2.GetMessageDataPointer(hMessage:= hMsg,peError:=ADR(ReadErr));	
			MsgID := cl2.GetMessageId(hMessage := hMsg, peError := ADR(ReadErr));
			proc_screen_data(MsgID := MsgID, pRxData := pRxData);
			cl2.FreeMessage(hMsg);		
			nReceived := cl2.GetMsgCount(hReceiverId :=hRecver_screen, peError := ADR(ReadErr));	
		END_WHILE
		(*
		IF nReceived <> 0 THEN
			hMsg := cl2.Read(hReceiverId :=hRecver_screen,pctMsgLeft:=ADR(nAvailable),peError:=ADR(ReadErr));
			pRxData := cl2.GetMessageDataPointer(hMessage:= hMsg,peError:=ADR(ReadErr));	
			MsgID := cl2.GetMessageId(hMessage := hMsg, peError := ADR(ReadErr));
			proc_screen_data(MsgID := MsgID, pRxData := pRxData);
			cl2.FreeMessage(hMsg);
		END_IF	
		nReceived := cl2.GetMsgCount(hReceiverId :=hRecver_screen, peError := ADR(ReadErr));
		IF nReceived <> 0 THEN
			hMsg := cl2.Read(hReceiverId :=hRecver_screen,pctMsgLeft:=ADR(nAvailable),peError:=ADR(ReadErr));
			pRxData := cl2.GetMessageDataPointer(hMessage:= hMsg,peError:=ADR(ReadErr));	
			MsgID := cl2.GetMessageId(hMessage := hMsg, peError := ADR(ReadErr));
			proc_screen_data(MsgID := MsgID, pRxData := pRxData);
			cl2.FreeMessage(hMsg);
		END_IF	
		*)
		//与电机CAN通讯失败
        T_Motor_CAN_fault(IN:=m>100,PT:=T#1S);
		//与屏通讯失败
        T_Screen_CAN_fault(IN:=n>100,PT:=T#1S);		
		can_stat := 30;
		
		
	30: //send data 
		//send data to motor
		set_buf_0801EE2A();
		CAN_Send_MSG(hCan0, 16#0801EE2A, 8, CanWriteData);
		
		//send data to screen
		// 12帧数据一起发送，以后可以根据需要调整发送间隔
		set_buf_18004f07();
		CAN_Send_MSG(hCan0, 16#18004F07, 8, CanWriteData);	
		
		set_buf_18014f07();
		CAN_Send_MSG(hCan0, 16#18014F07, 8, CanWriteData);	
			
		set_buf_18024f07();
		CAN_Send_MSG(hCan0, 16#18024F07, 8, CanWriteData);	
		
		set_buf_18034f07();
		CAN_Send_MSG(hCan0, 16#18034F07, 8, CanWriteData);	
	
		set_buf_18044f07();
		CAN_Send_MSG(hCan0, 16#18044F07, 8, CanWriteData);			
		
		set_buf_18054f07();
		CAN_Send_MSG(hCan0, 16#18054F07, 8, CanWriteData);			
		
		set_buf_18064f07();
		CAN_Send_MSG(hCan0, 16#18064F07, 8, CanWriteData);	
		
		set_buf_18074f07();
		CAN_Send_MSG(hCan0, 16#18074F07, 8, CanWriteData);	
		
		set_buf_18084f07();
		CAN_Send_MSG(hCan0, 16#18084F07, 8, CanWriteData);	
		
		set_buf_18094f07();
		CAN_Send_MSG(hCan0, 16#18094F07, 8, CanWriteData);	

		set_buf_18104f07();
		CAN_Send_MSG(hCan0, 16#18104F07, 8, CanWriteData);	

		set_buf_18114f07();
		CAN_Send_MSG(hCan0, 16#18114F07, 8, CanWriteData);	
		
		set_buf_18124f07();
		CAN_Send_MSG(hCan0, 16#18124F07, 8, CanWriteData);

		set_buf_18134f07();
		CAN_Send_MSG(hCan0, 16#18134F07, 8, CanWriteData);

		set_buf_18144f07();
		CAN_Send_MSG(hCan0, 16#18144F07, 8, CanWriteData);
	
		can_stat := 20;
	
	
	100:   //error
END_CASE

METHOD set_buf_18004f07 : bool
VAR_INPUT
END_VAR

VAR
	tmp_byte : BYTE := 0;
	tmp_uint: UINT := 0;
END_VAR
tmp_byte := 0;
CanWriteData[0] := tmp_byte;

tmp_byte := 0;
tmp_byte.0 := FALSE;
tmp_byte.1 := Wastewater_full_Fault;//污水满故障
tmp_byte.2 := T_DI_oil_filter_block.Q;//回油过滤堵塞
tmp_byte.3 := T_DI_oil_level_low.Q;//液压油位低故障
tmp_byte.4 := s00byte1bit4_res;
tmp_byte.5 := T_DI_cleanwater_LOW.Q;//水箱缺水故障
tmp_byte.6 := s00byte1bit6_res;
tmp_byte.7 := DI_Rcar_fault;//倒车故障停机
CanWriteData[1] := tmp_byte;

tmp_byte := 0;
tmp_byte.0 := Wastewater_full_Fault1;//污水满故障停机
tmp_byte.1 := NOT DI_power_on;//电源故障
tmp_byte.2 := T_Pumpspeed_H.Q;//高压水泵超速报警
tmp_byte.3 := T_Pumpspeed_HH.Q;//高压水泵超速停止
tmp_byte.4 := TEST_ALM;//请关闭测试
tmp_byte.5 := RCAR_ALM;//正在倒车中提示
tmp_byte.6 := Motor_Work_ALM;//请先启动电机提示
tmp_byte.7 := Func_test_HMI;//测试打开
CanWriteData[2] := tmp_byte;

tmp_byte := 0;
tmp_byte.0 := T_DI_air_press_low.Q;//气路系统压力低
tmp_byte.1 := T_DI_Rcar.Q;//倒车
tmp_byte.2 := s00byte3bit2_res;
tmp_byte.3 := DO_Hpre_pump_noWork;//高压水泵未啮合
tmp_byte.4 := T_Chassis_SOC_LOW.Q;//底盘电量低停机
tmp_byte.5 := DI_Hpre_valve_noOpen;//高压吹净球阀未打开
tmp_byte.6 := DI_Totvalve_noOpen;//高压水路球阀未打开
tmp_byte.7 := DO_Box_Up_arm;//请先打开箱门
CanWriteData[3] := tmp_byte;

tmp_byte := 0;
tmp_byte.0 := fog_Spump_arm;//隔膜泵球阀未打开
tmp_byte.1 := T_fog_pump_press_noOk.Q;//隔膜泵压力不正常
tmp_byte.2 := Fault_STOP;//故障停机
tmp_byte.3 := DO_Box_Down_arm;//请先放下撑杆
tmp_byte.4 := T_DI_wastewater_full.Q;//主污水箱水满
tmp_byte.5 := Backup_power_Test_warn;//请先打开备用动力开关
tmp_byte.6 := T_Chassis_CAN_fault.Q;//底盘CAN通讯故障
tmp_byte.7 := T_Motor_CAN_fault.Q;//与电机CAN通讯故障
CanWriteData[4] := tmp_byte;

tmp_byte := 0;
tmp_byte.0 := T_auxiliary_warte_dif.Q;//辅污水箱水位不一致
tmp_byte.1 := T_DI_auxiliary1_warte_H.Q;//辅1污水箱水满
tmp_byte.2 := T_DI_auxiliary2_warte_H.Q;//辅2污水箱水满
tmp_byte.3 := T_water_overflow_noClose.Q;//水路卸荷阀未关闭故障
tmp_byte.4 := T_water_overflow_noOpen.Q;//水路卸荷阀未打开故障
tmp_byte.5 := DI_backup_power_open;//备用动力打开提示
tmp_byte.6 := Chassis_SOC_LOW;//底盘电量低压20%提示
tmp_byte.7 := High_voltage_noReady;//底盘未上高压提示
CanWriteData[5] := tmp_byte;

tmp_byte := 0;
tmp_byte.0 := (DI_cleanwater_LOW<3000);
tmp_byte.1 := DI_Totvalve_Open;
tmp_byte.2 := DI_box_door_close;
tmp_byte.3 := DI_Hpre_valve_open;
tmp_byte.4 := DI_air_press_low;
tmp_byte.5 := DI_wastewater_full;
tmp_byte.6 := DI_Rod_noDown;
tmp_byte.7 := DI_backup_power_open;
CanWriteData[6] := tmp_byte;

tmp_byte := 0;
tmp_byte.0 := DI_water_overflow;
tmp_byte.1 := FALSE;
tmp_byte.2 := FALSE;
tmp_byte.3 := FALSE;
tmp_byte.4 := DI_fog_pump_press_ok;
tmp_byte.5 := DI_oil_level_low;
tmp_byte.6 := DI_oil_filter_block;
tmp_byte.7 := FALSE;
CanWriteData[7] := tmp_byte;

set_buf_18004f07 := TRUE;
END_METHOD

METHOD set_buf_18074f07 : bool
VAR_INPUT
END_VAR

VAR
	tmp_byte : BYTE := 0;
	tmp_uint: UINT := 0;
END_VAR
tmp_byte := ANY_TO_BYTE(S_Pumpspeed_arm MOD 256);
CanWriteData[0] := tmp_byte;

tmp_byte := ANY_TO_BYTE(S_Pumpspeed_arm/256);
CanWriteData[1] := tmp_byte;

tmp_byte := ANY_TO_BYTE(S_Pumpspeed_stop MOD 256);
CanWriteData[2] := tmp_byte;

tmp_byte := ANY_TO_BYTE(S_Pumpspeed_stop/256);
CanWriteData[3] := tmp_byte;

tmp_byte := ANY_TO_BYTE(S_MAX_Speed MOD 256);
CanWriteData[4] := tmp_byte;

tmp_byte := ANY_TO_BYTE(S_MAX_Speed/256);
CanWriteData[5] := tmp_byte;

tmp_byte := ANY_TO_BYTE(S_Idle_Speed MOD 256);
CanWriteData[6] := tmp_byte;

tmp_byte := ANY_TO_BYTE(S_Idle_Speed/256);
CanWriteData[7] := tmp_byte;

set_buf_18074f07 := TRUE;
END_METHOD

METHOD get_buf_0c00074f : bool
VAR_INPUT
	pRxData :POINTER TO CL2I.DATA;
END_VAR

VAR
	tmp_byte : BYTE := 0;

END_VAR
tmp_byte := pRxData^[0];
HMI_Awashsweep := tmp_byte.0;
HMI_Lwashsweep := tmp_byte.1;
HMI_Rwashsweep:= tmp_byte.2;
HMI_Asweeproad := tmp_byte.3;
HMI_Lsweeproad := tmp_byte.4;
HMI_Rsweeproad := tmp_byte.5;
HMI_Acleanwash := tmp_byte.6;
HMI_Lcleanwash := tmp_byte.7;

tmp_byte := pRxData^[1];
HMI_Rcleanwash:= tmp_byte.0;
HMI_stop_sweep:= tmp_byte.1;
HMI_start_motor := tmp_byte.2;
HMI_stop_motor := tmp_byte.3;
HMI_Inc_Speed:= tmp_byte.4;
HMI_Dec_Speed:= tmp_byte.5;
HMI_Standard_speed := tmp_byte.6;
HMI_Strong_speed := tmp_byte.7;

tmp_byte := pRxData^[2];
HMI_Door_Close := tmp_byte.0;
HMI_Door_Open := tmp_byte.1;
HMI_Box_Up:= tmp_byte.2;
HMI_Box_Down:= tmp_byte.3;
HMI_fog_Spump:= tmp_byte.4;
HMI_selfclean := tmp_byte.5;
HMI_wastewater_pump := tmp_byte.6;
c00byte2bit7_res := tmp_byte.7;

tmp_byte := pRxData^[3];
HMI_Sweep_Hspd:= tmp_byte.0;
HMI_Sweep_Mspd:= tmp_byte.1;
HMI_Sweep_Lspd:= tmp_byte.2;
HMI_Hpre_wash := tmp_byte.3;
HMI_pointshoot_up := tmp_byte.4;
HMI_pointshoot_down := tmp_byte.5;
HMI_pointshoot_left := tmp_byte.6;
HMI_pointshoot_right := tmp_byte.7;

tmp_byte := pRxData^[4];
HMI_drain_start := tmp_byte.0;
HMI_drain_auto := tmp_byte.1;
HMI_drain_manual := tmp_byte.2;
HMI_Lrod_drain := tmp_byte.3;
HMI_Rrod_drain := tmp_byte.4;
HMI_Hpressure_drain := tmp_byte.5;
HMI_selfclean_drain := tmp_byte.6;
HMI_Suction_drain := tmp_byte.7;

tmp_byte := pRxData^[6];
HMI_func_test := tmp_byte.0;
HMI_replace_Sweep:= tmp_byte.1;
HMI_intelligent := tmp_byte.2;
HMI_cleanly := tmp_byte.3;
HMI_normal := tmp_byte.4;
HMI_dirty := tmp_byte.5;
	
get_buf_0c00074f := TRUE;
END_METHOD

METHOD proc_screen_data : bool
VAR_INPUT
	MsgID     : CL2I.COBID;	
	pRxData :POINTER TO CL2I.DATA;
END_VAR
CASE MsgID OF
	16#0C00074F:
		get_buf_0c00074f(pRxData);
	16#0C01074F:
		get_buf_0c01074f(pRxData);
	16#0C02074F:
		get_buf_0c02074f(pRxData);
	16#0C03074F:
		get_buf_0c03074f(pRxData);	
	16#0C04074F:
		get_buf_0c04074f(pRxData);	
	16#0C05074F:
		get_buf_0c05074f(pRxData);
	16#0C06074F:
		get_buf_0c06074f(pRxData);
	16#0C07074F:
		get_buf_0c07074f(pRxData);	
END_CASE
END_METHOD

METHOD set_buf_18104f07 : bool
VAR_INPUT
END_VAR

VAR
	tmp_byte : BYTE := 0;
	tmp_uint: UINT := 0;
END_VAR

tmp_byte := 0;
tmp_byte := tmp_byte + 0*1;
tmp_byte := tmp_byte + Motor_direction_cw*4;
tmp_byte := tmp_byte + Motor_mode*16;
tmp_byte := tmp_byte + Motor_stat*64;
CanWriteData[0] := tmp_byte;

tmp_byte := 0;
tmp_byte := tmp_byte + Motor_bus_low_voltage*1;
tmp_byte := tmp_byte + Motor_bus_high_voltage*4;
tmp_byte := tmp_byte + MOtor_ctrller_high_temp*16;
tmp_byte := tmp_byte + Motor_high_temp*64;
CanWriteData[1] := tmp_byte;

tmp_byte := 0;
tmp_byte := tmp_byte + Motor_igbt_fault*1;
tmp_byte := tmp_byte + Motor_overspeed*4;
tmp_byte := tmp_byte + Motor_comm_error*16;
tmp_byte := tmp_byte + Motor_short*64;
CanWriteData[2] := tmp_byte;

tmp_byte := 0;
tmp_byte := tmp_byte + Motor_overload*1;
tmp_byte := tmp_byte + Motor_selfcheck_fault*4;
tmp_byte := tmp_byte + Motor_low_voltage*16;
tmp_byte := tmp_byte + Motor_sensor_fault*64;
CanWriteData[3] := tmp_byte;
	

set_buf_18104f07 := TRUE;
END_METHOD

METHOD set_buf_0801EE2A : BOOL
VAR_INPUT
END_VAR

VAR
	tmp_byte : BYTE := 0;
	tmp_uint: UINT := 0;
END_VAR
tmp_byte := ANY_TO_BYTE(16#19 MOD 256);
CanWriteData[0] := tmp_byte;
tmp_byte := ANY_TO_BYTE(0/256);
CanWriteData[1] := tmp_byte;

tmp_byte := ANY_TO_BYTE(0 MOD 256);
CanWriteData[2] := tmp_byte;
tmp_byte := ANY_TO_BYTE(SETspeed_PID MOD 256);
CanWriteData[3] := tmp_byte;

tmp_byte := ANY_TO_BYTE(SETspeed_PID/256);
CanWriteData[4] := tmp_byte;
tmp_byte := ANY_TO_BYTE(0/256);
CanWriteData[5] := tmp_byte;

tmp_byte := ANY_TO_BYTE(0 MOD 256);
CanWriteData[6] := tmp_byte;
tmp_byte := ANY_TO_BYTE(0/256);
CanWriteData[7] := tmp_byte;

set_buf_0801EE2A := TRUE;
END_METHOD

METHOD get_buf_0C112AEE : BOOL
VAR_INPUT
	pRxData :POINTER TO CL2I.DATA;
END_VAR

VAR

END_VAR
Motor_real_torque_HMI := 256*ANY_TO_UINT(pRxData^[1]) + ANY_TO_UINT(pRxData^[0]);
Motor_real_speed_HMI :=  256*ANY_TO_UINT(pRxData^[3]) + ANY_TO_UINT(pRxData^[2]);
Motor_bus_voltage_HMI :=  256*ANY_TO_UINT(pRxData^[5]) + ANY_TO_UINT(pRxData^[4]);
Motor_phase_current_HMI :=  256*ANY_TO_UINT(pRxData^[7]) + ANY_TO_UINT(pRxData^[6]);

get_buf_0C112AEE := TRUE;
END_METHOD

METHOD set_buf_18114f07 : bool
VAR_INPUT
END_VAR

VAR
	tmp_byte : BYTE := 0;
	tmp_uint: UINT := 0;
END_VAR
//tmp_byte := ANY_TO_BYTE(s09byte23_max_brake_torque/256);
//CanWriteData[3] := tmp_byte;

CanWriteData[0] := Chassis_Soc;//底盘电量
//CanWriteData[1] := s11byte0_chassis_power_percent;

tmp_byte := ANY_TO_BYTE(SETspeed_PID MOD 256);
CanWriteData[2] := tmp_byte;//设定电机转速
tmp_byte := ANY_TO_BYTE(SETspeed_PID/256);
CanWriteData[3] := tmp_byte;

tmp_byte := ANY_TO_BYTE(16#201 MOD 256);
CanWriteData[4] := tmp_byte;//程序版本
tmp_byte := ANY_TO_BYTE(16#201/256);
CanWriteData[5] := tmp_byte;

tmp_byte :=ANY_TO_BYTE(Chassis_speed MOD 256);// ANY_TO_BYTE(Chassis_speed MOD 256);
CanWriteData[6] := tmp_byte;//底盘车速
tmp_byte :=ANY_TO_BYTE(Chassis_speed/256); //ANY_TO_BYTE(Chassis_speed/256);
CanWriteData[7] := tmp_byte;

set_buf_18114f07 := TRUE;
END_METHOD

METHOD set_buf_18044f07 : bool
VAR_INPUT
END_VAR

VAR
	tmp_byte : BYTE := 0;
	tmp_uint: UINT := 0;
END_VAR

tmp_byte := 0;
tmp_byte.0 := Pointshoot_up_HMI;
tmp_byte.1 := Pointshoot_down_HMI;
tmp_byte.2 := Pointshoot_left_HMI;
tmp_byte.3 := Pointshoot_right_HMI;
tmp_byte.4 := Suction_drain_HMI;
tmp_byte.5 := FALSE;
tmp_byte.6 := FALSE;
tmp_byte.7 := FALSE;
CanWriteData[0] := tmp_byte;

tmp_byte := 0;
tmp_byte.0 := FALSE;
tmp_byte.1 := FALSE;
tmp_byte.2 := FALSE;
tmp_byte.3 := cooler_motor_Test;
tmp_byte.4 := cooler_fan_Test;
tmp_byte.5 := Sweep_Mspeed_Test;
tmp_byte.6 := Sweep_Lspeed_Test;
tmp_byte.7 := LSweep_Test;
CanWriteData[1] := tmp_byte;
	
tmp_byte := 0;
tmp_byte.0 := RSweep_Test;
tmp_byte.1 := ASweep_Test;
tmp_byte.2 := Box_Down_Test;
tmp_byte.3 := Box_Up_Test;
tmp_byte.4 := Suction_Down_Test;
tmp_byte.5 := Suction_Up_Test;
tmp_byte.6 := Boxdoor_open_Test;
tmp_byte.7 := Boxdoor_close_Test;
CanWriteData[2] := tmp_byte;

	
tmp_byte := 0;
tmp_byte.0 := LSweep_Down_Test;
tmp_byte.1 := LSweep_Up_Test;
tmp_byte.2 := RSweep_Down_Test;
tmp_byte.3 := RSweep_Up_Test;
tmp_byte.4 := Lrod_OUT_Test;
tmp_byte.5 := Rrod_OUT_Test;
tmp_byte.6 := Lrod_water_Test;
tmp_byte.7 := Rrod_water_Test;
CanWriteData[3] := tmp_byte;
	
tmp_byte := 0;
tmp_byte.0 := Suction_water_Test;
tmp_byte.1 := Hpre_wash_Test;
tmp_byte.2 := selfclean_water_Test;
tmp_byte.3 := Hpress_pump_gearin_Test;
tmp_byte.4 := Fog_pump_Test;
tmp_byte.5 := LSweep_out_Test;
tmp_byte.6 := RSweep_out_Test;
tmp_byte.7 := Wastewater_pump_Test;
CanWriteData[4] := tmp_byte;

tmp_byte := 0;
tmp_byte.0 := Wastewater_valve_Test;
tmp_byte.1 := Backup_power_Test;
tmp_byte.2 := Pointshoot_up_Test;
tmp_byte.3 := Pointshoot_down_Test;
tmp_byte.4 := Pointshoot_left_Test;
tmp_byte.5 := Pointshoot_right_Test;
tmp_byte.6 := Motor_Work;
tmp_byte.7 := SYS_work;
CanWriteData[5] := tmp_byte;

set_buf_18044f07 := TRUE;
END_METHOD

METHOD set_buf_18024f07 : bool
VAR_INPUT
END_VAR

VAR
	tmp_byte : BYTE := 0;
	tmp_uint: UINT := 0;
	
END_VAR
tmp_byte := 0;
tmp_byte.0:=DO_Lsweep_down_short;
tmp_byte.1:=DO_Lsweep_down_open;
tmp_byte.2:=DO_Lsweep_up_short;
tmp_byte.3:=DO_Lsweep_up_open;
tmp_byte.4:=DO_Rsweep_down_short;
tmp_byte.5:=DO_Rsweep_down_open;
tmp_byte.6:=DO_Rsweep_up_short;
tmp_byte.7:=DO_Rsweep_up_open;
CanWriteData[0] := tmp_byte;

tmp_byte := 0;
tmp_byte.0:=DO_Lsweep_out_short;
tmp_byte.1:=DO_Lsweep_out_open;
tmp_byte.2:=DO_Rsweep_out_short;
tmp_byte.3:=DO_Rsweep_out_open;
tmp_byte.4:=DO_Lrod_out_short;
tmp_byte.5:=DO_Lrod_out_open;
tmp_byte.6:=DO_Rrod_out_short;
tmp_byte.7:=DO_Rrod_out_open;
CanWriteData[1] := tmp_byte;

tmp_byte := 0;
tmp_byte.0:=DO_pointshoot_up_short;
tmp_byte.1:=DO_pointshoot_up_open;
tmp_byte.2:=DO_pointshoot_Down_short;
tmp_byte.3:=DO_pointshoot_Down_open;
tmp_byte.4:=DO_pointshoot_left_short;
tmp_byte.5:=DO_pointshoot_left_open;
tmp_byte.6:=DO_pointshoot_right_short;
tmp_byte.7:=DO_pointshoot_right_open;
CanWriteData[2] := tmp_byte;

tmp_byte := 0;
//tmp_byte.0:=;
//tmp_byte.1:=;
tmp_byte.2:=DO_water_overflow_short;
tmp_byte.3:=DO_water_overflow_open;
tmp_byte.4:=DO_Lrod_water_short;
tmp_byte.5:=DO_Lrod_water_open;
tmp_byte.6:=DO_Rrod_water_short;
tmp_byte.7:=DO_Rrod_water_open;
CanWriteData[3] := tmp_byte;

tmp_byte := 0;
tmp_byte.0:=DO_Suction_water_short;
tmp_byte.1:=DO_Suction_water_open;
tmp_byte.2:=DO_Hpressure_water_short;
tmp_byte.3:=DO_Hpressure_water_open;
tmp_byte.4:=DO_selfclean_water_short;
tmp_byte.5:=DO_selfclean_water_open;
tmp_byte.6:=DO_Hpre_pump_short;
tmp_byte.7:=DO_Hpre_pump_open;
CanWriteData[4] := tmp_byte;

tmp_byte := 0;
tmp_byte.0:=DO_fog_Spump_short;
tmp_byte.1:=DO_fog_Spump_open;
tmp_byte.2:=DO_Motor_en_short;
tmp_byte.3:=DO_Motor_en_open;
tmp_byte.4:=DO_watercooler_pump_short;
tmp_byte.5:=DO_watercooler_pump_open;
tmp_byte.6:=DO_cooler_fan_short;
tmp_byte.7:=DO_cooler_fan_open;
CanWriteData[5] := tmp_byte;

tmp_byte := 0;
tmp_byte.0:=DO_backup_power_short;
tmp_byte.1:=DO_backup_power_open;
//tmp_byte.2:=;
//tmp_byte.3:=;
//tmp_byte.4:=;
//tmp_byte.5:=;
//tmp_byte.6:=;
//tmp_byte.7:=;
CanWriteData[6] := tmp_byte;

tmp_byte := 0;
(*
tmp_byte.0:=;
tmp_byte.1:=;
tmp_byte.2:=;
tmp_byte.3:=;
tmp_byte.4:=;
tmp_byte.5:=;
tmp_byte.6:=;
tmp_byte.7:=;
*)
CanWriteData[7] := tmp_byte;
	
set_buf_18024f07 := TRUE;
END_METHOD

METHOD set_buf_18014f07 : bool
VAR_INPUT
END_VAR

VAR
	tmp_byte : BYTE := 0;
	tmp_uint: UINT := 0;
END_VAR
tmp_byte := 0;
tmp_byte.0 := DI_power_on;
tmp_byte.1 := DI_Rcar;
tmp_byte.2 := DI_oil_release_valve;
tmp_byte.3 := FALSE;
tmp_byte.4 := DI_auxiliary1_warte_H;
tmp_byte.5 := DI_auxiliary2_warte_H;
tmp_byte.6 := DI_Sweep_Up;
tmp_byte.7 := DI_Sweep_Down;
CanWriteData[0] := tmp_byte;

tmp_byte := 0;
tmp_byte.0 := DI_sweep_out;//s01byte1bit0_box_down;
tmp_byte.1 := DI_sweep_return;//s01byte1bit1_box_up;
tmp_byte.2 := FALSE;//s01byte1bit2_sucker_down;
tmp_byte.3 := FALSE;//s01byte1bit3_sucker_up;
tmp_byte.4 := FALSE;//s01byte1bit4_boxdoor_close;
tmp_byte.5 := FALSE;//s01byte1bit5_boxdoor_open;
tmp_byte.6 := FALSE;//s01byte1bit6_shooter_out;
tmp_byte.7 := FALSE;//s01byte1bit7_shooter_return;
CanWriteData[1] := tmp_byte;

tmp_byte := 0;
tmp_byte.0 :=  FALSE;//s01byte2bit0_right_sweeper_up;
tmp_byte.1 :=  FALSE;//s01byte2bit1_right_sweeper_down;
tmp_byte.2 :=  FALSE;//s01byte2bit2_cleanwater_high;
tmp_byte.3 := FALSE;// s01byte2bit3_alterable_box_low;
tmp_byte.4 := FALSE;// s01byte2bit4_res;
tmp_byte.5 := FALSE;
tmp_byte.6 := FALSE;
tmp_byte.7 := FALSE;
CanWriteData[2] := tmp_byte;

tmp_byte := 0;
tmp_byte.0 := DO_Lsweep_down;
tmp_byte.1 := DO_Lsweep_up;
tmp_byte.2 := DO_Rsweep_down;
tmp_byte.3 := DO_Rsweep_up;
tmp_byte.4 := DO_Lsweep_out;
tmp_byte.5 := DO_Rsweep_out;
tmp_byte.6 := DO_Lrod_out;
tmp_byte.7 := DO_Rrod_out;
CanWriteData[3] := tmp_byte;

tmp_byte := 0;
tmp_byte.0 :=  DO_pointshoot_up;
tmp_byte.1 :=  DO_pointshoot_down;
tmp_byte.2 :=  DO_pointshoot_left;
tmp_byte.3 :=  DO_pointshoot_right;
tmp_byte.4 :=  FALSE;//s01byte4bit4_oil_release_valve;//
tmp_byte.5 := DO_water_overflow;
tmp_byte.6 := DO_Lrod_water;
tmp_byte.7 := DO_Rrod_water;
CanWriteData[4] := tmp_byte;


tmp_byte := 0;
tmp_byte.0 := DO_Suction_water;
tmp_byte.1 := DO_Hpressure_water;
tmp_byte.2 := DO_selfclean_water;
tmp_byte.3 := DO_Hpre_pump;
tmp_byte.4 := DO_fog_Spump;
tmp_byte.5 := DO_Motor_en;
tmp_byte.6 := DO_watercooler_pump;
tmp_byte.7 := DO_cooler_fan;
CanWriteData[5] := tmp_byte;


tmp_byte := 0;
tmp_byte.0 := DO_backup_power;
tmp_byte.1 := DO_wastewater_valve;
tmp_byte.2 := DO_wastewater_pump;
tmp_byte.3 := DO_oil_release_valve;
tmp_byte.4 := DO_Sweep_Mspeed;
tmp_byte.5 := DO_Sweep_Lspeed;
tmp_byte.6 := DO_RSweep;
tmp_byte.7 := DO_LASweep;
CanWriteData[6] := tmp_byte;

tmp_byte := 0;
tmp_byte.0 := DO_RASweep;
tmp_byte.1 := DO_Box_Down;
tmp_byte.2 := DO_Box_Up;
tmp_byte.3 := DO_Suction_Down;
tmp_byte.4 := DO_Suction_Up;
tmp_byte.5 := DO_Door_Open;
tmp_byte.6 := DO_Door_Close;
tmp_byte.7 := FALSE;
CanWriteData[7] := tmp_byte;

set_buf_18014f07 := TRUE;
END_METHOD

METHOD get_buf_0c02074f : bool
VAR_INPUT
	pRxData :POINTER TO CL2I.DATA;
END_VAR

VAR
	tmp_byte : BYTE := 0;
	tmp_uint: UINT := 0;
END_VAR

Re_IncDec_Speed:= 256*ANY_TO_UINT(pRxData^[5]) + ANY_TO_UINT(pRxData^[4]);
Re_motor_min_speed := 256*ANY_TO_UINT(pRxData^[7]) + ANY_TO_UINT(pRxData^[6]);

get_buf_0c02074f := TRUE;
END_METHOD

METHOD get_buf_0C132AEE : BOOL
VAR_INPUT
	pRxData :POINTER TO CL2I.DATA;
END_VAR

VAR
	tmp_byte : BYTE := 0;
	tmp_uint: UINT := 0;
END_VAR
Motor_direction_cw := ANY_TO_BYTE(pRxData^[0]/4)MOD 4;
Motor_mode := ANY_TO_BYTE(pRxData^[0]/16) MOD 4;
Motor_stat := ANY_TO_BYTE(pRxData^[0]/64)MOD 4;

Motor_bus_low_voltage := ANY_TO_BYTE(pRxData^[1]/1)MOD 4;
Motor_bus_high_voltage := ANY_TO_BYTE(pRxData^[1]/4)MOD 4;
MOtor_ctrller_high_temp := ANY_TO_BYTE(pRxData^[1]/16)MOD 4;
Motor_high_temp := ANY_TO_BYTE(pRxData^[1]/64)MOD 4;

Motor_igbt_fault := ANY_TO_BYTE(pRxData^[2]/1)MOD 4;
Motor_overspeed := ANY_TO_BYTE(pRxData^[2]/4)MOD 4;
Motor_comm_error := ANY_TO_BYTE(pRxData^[2]/16)MOD 4;
Motor_short := ANY_TO_BYTE(pRxData^[2]/64)MOD 4;

Motor_overload := ANY_TO_BYTE(pRxData^[3]/1)MOD 4;
Motor_selfcheck_fault := ANY_TO_BYTE(pRxData^[3]/4)MOD 4;
Motor_low_voltage := ANY_TO_BYTE(pRxData^[3]/16)MOD 4;
Motor_sensor_fault := ANY_TO_BYTE(pRxData^[3]/64)MOD 4;


get_buf_0C132AEE := TRUE;
END_METHOD

METHOD get_buf_0c05074f : bool
VAR_INPUT
	pRxData :POINTER TO CL2I.DATA;
END_VAR

Re_clean_low_speed := 256*ANY_TO_UINT(pRxData^[1]) + ANY_TO_UINT(pRxData^[0]);
Re_clean_midlow_speed := 256*ANY_TO_UINT(pRxData^[3]) + ANY_TO_UINT(pRxData^[2]);
Re_clean_midhigh_speed := 256*ANY_TO_UINT(pRxData^[5]) + ANY_TO_UINT(pRxData^[4]);
Re_clean_high_speed := 256*ANY_TO_UINT(pRxData^[7]) + ANY_TO_UINT(pRxData^[6]);

get_buf_0c05074f := TRUE;
END_METHOD

METHOD get_buf_0c04074f : bool
VAR_INPUT
	pRxData :POINTER TO CL2I.DATA;
END_VAR

Re_Pumpspeed_arm:= 256*ANY_TO_UINT(pRxData^[1]) + ANY_TO_UINT(pRxData^[0]);
Re_Pumpspeed_stop:= 256*ANY_TO_UINT(pRxData^[3]) + ANY_TO_UINT(pRxData^[2]);
Re_MAX_Speed:= 256*ANY_TO_UINT(pRxData^[5]) + ANY_TO_UINT(pRxData^[4]);
Re_Idle_Speed := 256*ANY_TO_UINT(pRxData^[7]) + ANY_TO_UINT(pRxData^[6]);

get_buf_0c04074f := TRUE;
END_METHOD

METHOD set_buf_18054f07 : bool
VAR_INPUT
END_VAR

VAR
	tmp_byte : BYTE := 0;
	tmp_uint: UINT := 0;
END_VAR
tmp_byte := ANY_TO_BYTE(S_IncDec_Speed MOD 256);
CanWriteData[4] := tmp_byte;

tmp_byte := ANY_TO_BYTE(S_IncDec_Speed/256);
CanWriteData[5] := tmp_byte;

tmp_byte := ANY_TO_BYTE(S_min_speed MOD 256);
CanWriteData[6] := tmp_byte;

tmp_byte := ANY_TO_BYTE(S_min_speed/256);
CanWriteData[7] := tmp_byte;

set_buf_18054f07 := TRUE;
END_METHOD

METHOD get_buf_0c01074f : bool
VAR_INPUT
	pRxData :POINTER TO CL2I.DATA;
END_VAR

VAR
	tmp_byte : BYTE := 0;
	tmp_uint: UINT := 0;
END_VAR
tmp_byte := pRxData^[0];
Test_watercooler_pump := tmp_byte.3;
Test_cooler_fan := tmp_byte.4;

tmp_byte := pRxData^[1];
Test_Sweep_Mspeed:= tmp_byte.0;
Test_Sweep_Lspeed:= tmp_byte.1;
Test_LSweep:= tmp_byte.2;
Test_RSweep:= tmp_byte.3;
Test_ASweep:= tmp_byte.4;
Test_Box_Down:= tmp_byte.5;
Test_Box_Up:= tmp_byte.6;
Test_Suction_Down:= tmp_byte.7;

tmp_byte := pRxData^[2];
Test_Suction_Up:= tmp_byte.0;
Test_Door_Open:= tmp_byte.1;
Test_Door_Close:= tmp_byte.2;
Test_LSweep_Down:= tmp_byte.6;
Test_LSweep_Up:= tmp_byte.7;

tmp_byte := pRxData^[3];
Test_RSweep_Down:= tmp_byte.0;
Test_RSweep_Up:= tmp_byte.1;
Test_LSweep_out := tmp_byte.2;
Test_RSweep_out := tmp_byte.3;
Test_Lrod_OUT:= tmp_byte.4;
Test_Rrod_OUT:= tmp_byte.5;
Test_Lrod_water:= tmp_byte.6;
Test_Rrod_water:= tmp_byte.7;

tmp_byte := pRxData^[4];
Test_Suction_water:= tmp_byte.0;
Test_Hpre_wash:= tmp_byte.1;
Test_selfclean:= tmp_byte.2;
Test_Hpre_pump_gearin := tmp_byte.3;
Test_fogpump := tmp_byte.4;
Test_pointshoot_up := tmp_byte.5;
Test_pointshoot_down := tmp_byte.6;
Test_pointshoot_left := tmp_byte.7;

tmp_byte := pRxData^[5];
Test_pointshoot_right := tmp_byte.0;
Test_wastewater_pump := tmp_byte.2;
Test_wastewater_valve := tmp_byte.3;

tmp_byte := pRxData^[6];
Test_backup_power := tmp_byte.0;

get_buf_0c01074f := TRUE;
END_METHOD

METHOD get_buf_0C122AEE : BOOL
VAR_INPUT
	pRxData :POINTER TO CL2I.DATA;
END_VAR

VAR
	tmp_byte : BYTE := 0;
	tmp_uint: UINT := 0;
END_VAR
Motor_max_dirve_torque_HMI := 256*ANY_TO_UINT(pRxData^[1]) + ANY_TO_UINT(pRxData^[0]);
Motor_max_brake_torque_HMI :=  256*ANY_TO_UINT(pRxData^[3]) + ANY_TO_UINT(pRxData^[2]);
Motor_temp_controller_HMI  := ANY_TO_BYTE(pRxData^[4]);
Motor_temp_HMI  := ANY_TO_BYTE(pRxData^[5]);

Motor_max_speed_HMI :=  256*ANY_TO_UINT(pRxData^[7]) + ANY_TO_UINT(pRxData^[6]);

get_buf_0C122AEE := TRUE;
END_METHOD

METHOD set_buf_18124f07 : BOOL
VAR_INPUT
END_VAR

VAR
	tmp_byte : BYTE := 0;
	tmp_uint: UINT := 0;
END_VAR

tmp_byte := ANY_TO_BYTE(S_clean_low_speed MOD 256);
CanWriteData[0] := tmp_byte;
tmp_byte := ANY_TO_BYTE(S_clean_low_speed/256);
CanWriteData[1] := tmp_byte;

tmp_byte := ANY_TO_BYTE(S_clean_midlow_speed MOD 256);
CanWriteData[2] := tmp_byte;
tmp_byte := ANY_TO_BYTE(S_clean_midlow_speed/256);
CanWriteData[3] := tmp_byte;

tmp_byte := ANY_TO_BYTE(S_clean_midhigh_speed MOD 256);
CanWriteData[4] := tmp_byte;
tmp_byte := ANY_TO_BYTE(S_clean_midhigh_speed/256);
CanWriteData[5] := tmp_byte;

tmp_byte := ANY_TO_BYTE(S_clean_high_speed MOD 256);
CanWriteData[6] := tmp_byte;
tmp_byte := ANY_TO_BYTE(S_clean_high_speed/256);
CanWriteData[7] := tmp_byte;

set_buf_18124f07 := TRUE;
END_METHOD

METHOD set_buf_18084f07 : bool
VAR_INPUT
END_VAR

VAR
	tmp_byte : BYTE := 0;
	tmp_uint: UINT := 0;
END_VAR
tmp_byte := ANY_TO_BYTE(Motor_real_torque_HMI MOD 256);
CanWriteData[0] := tmp_byte;

tmp_byte := ANY_TO_BYTE(Motor_real_torque_HMI/256);
CanWriteData[1] := tmp_byte;

IF Motor_real_speed_HMI<5 THEN
   Motor_real_speed_HMI:=0;
   ELSE
	Motor_real_speed_HMI:=Motor_real_speed_HMI;   
END_IF
                 
tmp_byte := ANY_TO_BYTE(Motor_real_speed_HMI MOD 256);
CanWriteData[2] := tmp_byte;

tmp_byte := ANY_TO_BYTE(Motor_real_speed_HMI/256);
CanWriteData[3] := tmp_byte;

tmp_byte := ANY_TO_BYTE(Motor_bus_voltage_HMI MOD 256);
CanWriteData[4] := tmp_byte;

tmp_byte := ANY_TO_BYTE(Motor_bus_voltage_HMI/256);
CanWriteData[5] := tmp_byte;

tmp_byte := ANY_TO_BYTE(Motor_phase_current_HMI MOD 256);
CanWriteData[6] := tmp_byte;

tmp_byte := ANY_TO_BYTE(Motor_phase_current_HMI/256);
CanWriteData[7] := tmp_byte;


set_buf_18084f07 := TRUE;
END_METHOD

METHOD set_buf_18064f07 : bool
VAR_INPUT
END_VAR


VAR
	tmp_byte : BYTE := 0;
	tmp_uint: UINT := 0;
END_VAR

tmp_byte := ANY_TO_BYTE(S_Standard_Speed MOD 256);
CanWriteData[0] := tmp_byte;

tmp_byte := ANY_TO_BYTE(S_Standard_Speed/256);
CanWriteData[1] := tmp_byte;

tmp_byte := ANY_TO_BYTE(S_Strong_Speed MOD 256);
CanWriteData[2] := tmp_byte;

tmp_byte := ANY_TO_BYTE(S_Strong_Speed/256);
CanWriteData[3] := tmp_byte;

tmp_byte := ANY_TO_BYTE(S_Sweep_Speed MOD 256);
CanWriteData[4] := tmp_byte;

tmp_byte := ANY_TO_BYTE(S_Sweep_Speed/256);
CanWriteData[5] := tmp_byte;

set_buf_18064f07 := TRUE;
END_METHOD

METHOD set_buf_18144f07 : BOOL
VAR_INPUT
END_VAR

VAR
	tmp_byte : BYTE := 0;
	tmp_uint: UINT := 0;
END_VAR

tmp_byte := ANY_TO_BYTE(S_dirty_low_speed MOD 256);
CanWriteData[0] := tmp_byte;
tmp_byte := ANY_TO_BYTE(S_dirty_low_speed/256);
CanWriteData[1] := tmp_byte;

tmp_byte := ANY_TO_BYTE(S_dirty_midlow_speed MOD 256);
CanWriteData[2] := tmp_byte;
tmp_byte := ANY_TO_BYTE(S_dirty_midlow_speed/256);
CanWriteData[3] := tmp_byte;

tmp_byte := ANY_TO_BYTE(S_dirty_midhigh_speed MOD 256);
CanWriteData[4] := tmp_byte;
tmp_byte := ANY_TO_BYTE(S_dirty_midhigh_speed/256);
CanWriteData[5] := tmp_byte;

tmp_byte := ANY_TO_BYTE(S_dirty_high_speed MOD 256);
CanWriteData[6] := tmp_byte;
tmp_byte := ANY_TO_BYTE(S_dirty_high_speed/256);
CanWriteData[7] := tmp_byte;

set_buf_18144f07 := TRUE;
END_METHOD

METHOD set_buf_18094f07 : bool
VAR_INPUT
END_VAR

VAR
	tmp_byte : BYTE := 0;
	tmp_uint: UINT := 0;
END_VAR

tmp_byte := ANY_TO_BYTE(Motor_max_dirve_torque_HMI MOD 256);
CanWriteData[0] := tmp_byte;

tmp_byte := ANY_TO_BYTE(Motor_max_dirve_torque_HMI/256);
CanWriteData[1] := tmp_byte;

tmp_byte := ANY_TO_BYTE(Motor_max_brake_torque_HMI MOD 256);
CanWriteData[2] := tmp_byte;

tmp_byte := ANY_TO_BYTE(Motor_max_brake_torque_HMI/256);
CanWriteData[3] := tmp_byte;

tmp_byte := Motor_temp_controller_HMI;
CanWriteData[4] := tmp_byte;

tmp_byte := Motor_temp_HMI;
CanWriteData[5] := tmp_byte;

tmp_byte := ANY_TO_BYTE(Motor_max_speed_HMI MOD 256);
CanWriteData[6] := tmp_byte;

tmp_byte := ANY_TO_BYTE(Motor_max_speed_HMI/256);
CanWriteData[7] := tmp_byte;

set_buf_18094f07 := TRUE;
END_METHOD

METHOD set_buf_18034f07 : bool
VAR_INPUT
END_VAR

VAR
	tmp_byte : BYTE := 0;
	tmp_uint: UINT := 0;
END_VAR

tmp_byte := 0;
//tmp_byte := tmp_byte + s03byte0bit01_res*1;
//tmp_byte := tmp_byte + s03byte0bit23_water_coller_motor*4;
//tmp_byte := tmp_byte + s03byte0bit45_cooler_fan*16;
//tmp_byte := tmp_byte + s03byte0bit67_lowpress_pump*64;
CanWriteData[0] := tmp_byte;

tmp_byte := 0;
CanWriteData[1] := tmp_byte;

tmp_byte := 0;
CanWriteData[2] := tmp_byte;

tmp_byte := 0;
tmp_byte.0 := AwashSweep_HMI;
tmp_byte.1 := LwashSweep_HMI;
tmp_byte.2 := RwashSweep_HMI;
tmp_byte.3 := ASweeproad_HMI;
tmp_byte.4 := LSweeproad_HMI;
tmp_byte.5 := RSweeproad_HMI;
tmp_byte.6 := Aclean_HMI;
tmp_byte.7 := Lclean_HMI;
CanWriteData[3] := tmp_byte;
	
tmp_byte := 0;
tmp_byte.0 := Rclean_HMI;
tmp_byte.1 := Sweep_stop_HMI;
tmp_byte.2 := DO_fog_Spump1;
tmp_byte.3 := DO_selfclean_water1;
tmp_byte.4 := DO_Door_Close1;
tmp_byte.5 := DO_Door_Open1;
tmp_byte.6 := DO_Box_Up1;
tmp_byte.7 := DO_Box_Down1;
CanWriteData[4] := tmp_byte;

tmp_byte := 0;
//tmp_byte.0 := s03byte5bit0_motor_start;
//tmp_byte.1 := s03byte5bit1_motor_stop;
//tmp_byte.2 := motor_work;
//tmp_byte.3 := FALSE;
tmp_byte.4 := Standard_speed_HMI;
tmp_byte.5 := Strong_speed_HMI;
tmp_byte.6 := Sweep_HSpeed_HMI;
tmp_byte.7 := Sweep_MSpeed_HMI;
CanWriteData[5] := tmp_byte;

tmp_byte := 0;
tmp_byte.0 := Sweep_LSpeed_HMI;
tmp_byte.1 := DO_Hpressure_water1;
tmp_byte.2 := Drain_start_HMI;
tmp_byte.3 := Drain_auto_HMI;
tmp_byte.4 := Drain_manual_HMI;
tmp_byte.5 := Lrod_drain_HMI;
tmp_byte.6 := Rrod_drain_HMI;
tmp_byte.7 := Hpressure_drain_HMI;
CanWriteData[6] := tmp_byte;

tmp_byte := 0;
tmp_byte.0 := Selfclean_drain_HMI;
tmp_byte.1 := replace_Sweep_HMI;
tmp_byte.2 := Func_test_HMI;
tmp_byte.3 := Intelligent_HMI;
tmp_byte.4 := Cleanly_HMI;
tmp_byte.5 := Normal_HMI;
tmp_byte.6 := Dirty_HMI;
tmp_byte.7 := DO_wastewater_pump_open1;
CanWriteData[7] := tmp_byte;

set_buf_18034f07 := TRUE;
END_METHOD

METHOD set_buf_18134f07 : BOOL
VAR_INPUT
END_VAR

VAR
	tmp_byte : BYTE := 0;
	tmp_uint: UINT := 0;
END_VAR

tmp_byte := ANY_TO_BYTE(S_normal_low_speed MOD 256);
CanWriteData[0] := tmp_byte;
tmp_byte := ANY_TO_BYTE(S_normal_low_speed/256);
CanWriteData[1] := tmp_byte;

tmp_byte := ANY_TO_BYTE(S_normal_midlow_speed MOD 256);
CanWriteData[2] := tmp_byte;
tmp_byte := ANY_TO_BYTE(S_normal_midlow_speed/256);
CanWriteData[3] := tmp_byte;

tmp_byte := ANY_TO_BYTE(S_normal_midhigh_speed MOD 256);
CanWriteData[4] := tmp_byte;
tmp_byte := ANY_TO_BYTE(S_normal_midhigh_speed/256);
CanWriteData[5] := tmp_byte;

tmp_byte := ANY_TO_BYTE(S_normal_high_speed MOD 256);
CanWriteData[6] := tmp_byte;
tmp_byte := ANY_TO_BYTE(S_normal_high_speed/256);
CanWriteData[7] := tmp_byte;

set_buf_18134f07 := TRUE;
END_METHOD

METHOD get_buf_0c03074f : bool
VAR_INPUT
	pRxData :POINTER TO CL2I.DATA;
END_VAR

Re_normal_speed := 256*ANY_TO_UINT(pRxData^[1]) + ANY_TO_UINT(pRxData^[0]);
Re_strong_Speed:= 256*ANY_TO_UINT(pRxData^[3]) + ANY_TO_UINT(pRxData^[2]);
Re_Sweep_Speed:= 256*ANY_TO_UINT(pRxData^[5]) + ANY_TO_UINT(pRxData^[4]);

get_buf_0c03074f := TRUE;
END_METHOD

METHOD get_buf_0c07074f : bool
VAR_INPUT
	pRxData :POINTER TO CL2I.DATA;
END_VAR

Re_dirty_low_speed := 256*ANY_TO_UINT(pRxData^[1]) + ANY_TO_UINT(pRxData^[0]);
Re_dirty_midlow_speed := 256*ANY_TO_UINT(pRxData^[3]) + ANY_TO_UINT(pRxData^[2]);
Re_dirty_midhigh_speed := 256*ANY_TO_UINT(pRxData^[5]) + ANY_TO_UINT(pRxData^[4]);
Re_dirty_high_speed := 256*ANY_TO_UINT(pRxData^[7]) + ANY_TO_UINT(pRxData^[6]);

get_buf_0c07074f := TRUE;
END_METHOD

METHOD get_buf_0c06074f : bool
VAR_INPUT
	pRxData :POINTER TO CL2I.DATA;
END_VAR

Re_normal_low_speed := 256*ANY_TO_UINT(pRxData^[1]) + ANY_TO_UINT(pRxData^[0]);
Re_normal_midlow_speed := 256*ANY_TO_UINT(pRxData^[3]) + ANY_TO_UINT(pRxData^[2]);
Re_normal_midhigh_speed := 256*ANY_TO_UINT(pRxData^[5]) + ANY_TO_UINT(pRxData^[4]);
Re_normal_high_speed := 256*ANY_TO_UINT(pRxData^[7]) + ANY_TO_UINT(pRxData^[6]);

get_buf_0c06074f := TRUE;
END_METHOD

END_PROGRAM

// Changsha_Xiangji_ARM_Cortex_A9_xilinx_zynq7000_linux/Application/CAN_COMM/CAN_Send_MSG
FUNCTION CAN_Send_MSG : BOOL
VAR_INPUT
	h:	CAA.HANDLE;     //hCan
	TMsgID   : CL2I.COBID;
    TusiLen  : USINT;
	TData    : ARRAY[0..7] OF BYTE;    	
END_VAR
VAR
   Send:CAA.HANDLE;
   WriteErr   : CL2.ERROR;
   p_data:POINTER TO CL2I.DATA;
END_VAR

IF  (0=h) THEN
	RETURN;
END_IF 

Send := cl2.CreateMessage(hDriver := h,
                          cobID := TMsgID,
						  usiLength := TusiLen,
						  xRTR := FALSE,
						  x29BitID := TRUE,
						  peError := ADR(WriteErr));
						  
IF Send <> CAA.gc_hINVALID THEN
	p_data := cl2.GetMessageDataPointer(hMessage := Send,peError:=ADR(WriteErr));
	IF (WriteErr = CL2.ERROR.NO_ERROR) THEN
		SysMemCpy(pDest:=p_data,pSrc:=ADR(TData),udiCount:=SIZEOF(TData));
	END_IF
	
	WriteErr := cl2.Write(hDriver := h,hMessage:=Send,usiPriority:=1,xEnableSyncWindow:=FALSE);
	IF (WriteErr <> CL2.ERROR.NO_ERROR) THEN
        cl2.FreeMessage(hMessage:=Send);		
	END_IF
	
	p_data := CAA.gc_pNULL;
	Send:=CAA.gc_hINVALID;	
END_IF

END_FUNCTION

// Changsha_Xiangji_ARM_Cortex_A9_xilinx_zynq7000_linux/Application/CAN_COMM/prg_can1
PROGRAM prg_can1    //CAN1   与上装电机驱动器通信
VAR
	hCan1:CAA.HANDLE:=0;
    CanWriteData : ARRAY[0..7] OF BYTE;
    CanWriteMsgID:UDINT;
	CanReadData : ARRAY[0..7] OF BYTE;  
	CanReadMsgID:UDINT;
	bModifyTimeFlag :BOOL := FALSE;
	

	
	//通过CAN总线从驱动器读到的信息
	c11byte01_torque:UINT:= 0;
	c11byte23_speed:UINT:= 0;
	c11byte45_voltage:UINT:=0;
	c11byte67_current:UINT:= 0;
	
	c12byte01_drv_torque_max:UINT:= 0;
	c12byte23_brk_torque_max:UINT := 0;
	c12byte4_temp_controller:INT:= 0; //offset:  -40
	c12byte5_temp_motor:INT := 0;  //offset: -40
	c12byte67_speed_max:UINT:= 0;  
	
	c13byte0bit23_cw:BYTE:=0; //00:stop, 01:ccw,  10:cw
	c13byte0bit45_mode:BYTE := 01; //01:drive, 10:brake
	c13byte0bit67_stat:BYTE := 00; //00: enable, 01:running, 10:stop, 11:fault
	
	c13byte1bit01_low_vol:BYTE := 00; //00: normal, 01:warning, 10: fault
	c13byte1bit23_high_vol:BYTE := 0;
	c13byte1bit45_temp_ctrler:BYTE := 0;
	c13byte1bit67_temp_motor:BYTE := 0;
	
	c13byte2bit01_igbt:BYTE := 0;
	c13byte2bit23_speed:BYTE := 0;
	c13byte2bit45_comm:BYTE := 0;
	c13byte2bit67_short:BYTE := 0;
	
	c13byte3bit01_overload:BYTE := 0;
	c13byte3bit23_selfcheck:BYTE := 0;
	c13byte3bit45_low_voltage:BYTE := 0;
	c13byte3bit67_sensor:BYTE := 0;
	
	
	//发送给驱动器的信息
	byte0bit6_enable:BOOL := FALSE;
	byte0bit45_cw:BYTE := 01;  //01:CCW,  10:CW 方向
	byte0bit23_ctrl:BYTE := 01; //01:转矩， 10：转速
	byte0bit01_mode:BYTE := 01;  //01:牵引， 10: 制动
	byte12_torque:UINT:= 0; //转矩
	byte34_speed:UINT := 0;  //转速
	

	//底盘handle
	hReceiver_ready:CAA.HANDLE;
	hReceiver_speed:CAA.HANDLE;
	hReceiver_soc:CAA.HANDLE;

	tmp_byte:BYTE;
	tmp_uint:UINT;
	Err:CAA.ERROR;
	
	hMsg : CAA.HANDLE;
	nReceived : CAA.COUNT;
	nAvailable: CAA.COUNT;
	ReadErr   : CAA.ERROR;
	MsgID     : CL2I.COBID;	
	pRxData :POINTER TO CL2I.DATA;
	
	can_stat : DINT := 0;
	h: INT := 0;
	a: BOOL := FALSE;
	T_SOC_LOW: Ton;
END_VAR

CASE can_stat OF
	0:   //init can port0 and port1
		hCan1 := cl2.DriverOpenH(usiNetId:=1,uiBaudRate:=250,xSupport29Bits:=TRUE,ctMessages:=100,peError:=ADR(Err));	 //CAN1
		IF hCan1 > 0 THEN
			can_stat := 10;
		END_IF
	

	10: //create receiver for data
		//创建接收底盘信息的接收器: ID:0x18c21726,  byte6.bit2  READY灯	
	  	hReceiver_ready := CL2.CreateMaskReceiver(hDriver := hCan1,
			cobIdValue := 16#18C21726, //cobID value
			cobIdMask := 16#FFFFFFFF, //cobID mask ==> all bits of value are relevant									
			xRTRValue := FALSE, //no RTR messages
			xRTRMask := FALSE, //activate RTR filter ==> xRTRValue will be checked
			x29BitIdValue := TRUE, //29 bit CAN messages
			x29BitIdMask := TRUE, //activate 29 bit filter ==> x29BitIdValue will be checked
			xTransmitValue := FALSE, //only receive messages, no transmit message loopback
			xTransmitMask := FALSE, //activate transmit mask filter ==> xTransmitValue will be checked
			xAlwaysNewest := FALSE, //FALSE := receiver with queue; TRUE: only newest message
			eEvent := CB.EVENT.NO_EVENT,  //no receive event
			xEnableSyncWindow := FALSE, //not implemented
			peError := ADR(Err) //optional pointer to error
			);
		//创建接收底盘信息的接收器: ID:0x18c31726,  byte7  车速	
	  	hReceiver_speed := CL2.CreateMaskReceiver(hDriver := hCan1,
			cobIdValue := 16#18C31726, //cobID value
			cobIdMask := 16#FFFFFFFF, //cobID mask ==> all bits of value are relevant									
			xRTRValue := FALSE, //no RTR messages
			xRTRMask := FALSE, //activate RTR filter ==> xRTRValue will be checked
			x29BitIdValue := TRUE, //29 bit CAN messages
			x29BitIdMask := TRUE, //activate 29 bit filter ==> x29BitIdValue will be checked
			xTransmitValue := FALSE, //only receive messages, no transmit message loopback
			xTransmitMask := FALSE, //activate transmit mask filter ==> xTransmitValue will be checked
			xAlwaysNewest := FALSE, //FALSE := receiver with queue; TRUE: only newest message
			eEvent := CB.EVENT.NO_EVENT, //no receive event
			xEnableSyncWindow := FALSE, //not implemented
			peError := ADR(Err) //optional pointer to error
			);	
		
		//创建接收底盘信息的接收器: ID:0x182126f4,  byte0*0.4  剩余SOC百分比
		hReceiver_soc := CL2.CreateMaskReceiver(hDriver := hCan1,
			cobIdValue := 16#182126F4, //cobID value
			cobIdMask := 16#FFFFFFFF, //cobID mask ==> all bits of value are relevant									
			xRTRValue := FALSE, //no RTR messages
			xRTRMask := FALSE, //activate RTR filter ==> xRTRValue will be checked
			x29BitIdValue := TRUE, //no 29 bit CAN messages
			x29BitIdMask := TRUE, //activate 29 bit filter ==> x29BitIdValue will be checked
			xTransmitValue := FALSE, //only receive messages, no transmit message loopback
			xTransmitMask := FALSE, //activate transmit mask filter ==> xTransmitValue will be checked
			xAlwaysNewest := FALSE, //FALSE := receiver with queue; TRUE: only newest message
			eEvent := CB.EVENT.NO_EVENT, //no receive event
			xEnableSyncWindow := FALSE, //not implemented
			peError := ADR(Err) //optional pointer to error
		);

		
		IF (hReceiver_ready <> 0 AND hReceiver_speed <> 0 AND hReceiver_soc <> 0  ) THEN
			 can_stat := 20;
		ELSE
			RETURN;
		END_IF
	
	20:  //receive data
		//接收底盘信息: ID:0x18c21726,  byte6.bit2  READY灯	
		nReceived := cl2.GetMsgCount(hReceiverId :=hReceiver_ready, peError := ADR(ReadErr));
		WHILE nReceived > 0 DO
			hMsg := cl2.Read(hReceiverId :=hReceiver_ready,pctMsgLeft:=ADR(nAvailable),peError:=ADR(ReadErr));
			pRxData := cl2.GetMessageDataPointer(hMessage:= hMsg,peError:=ADR(ReadErr));	
			tmp_byte := pRxData^[6];
			High_voltage_Ready := tmp_byte.2;
			cl2.FreeMessage(hMsg);	
			nReceived := cl2.GetMsgCount(hReceiverId :=hReceiver_ready, peError := ADR(ReadErr));
		END_WHILE

		//接收底盘信息: ID:0x18c31726,  byte7  车速	
		nReceived := cl2.GetMsgCount(hReceiverId :=hReceiver_speed, peError := ADR(ReadErr));
		WHILE nReceived > 0 DO
			hMsg := cl2.Read(hReceiverId :=hReceiver_speed,pctMsgLeft:=ADR(nAvailable),peError:=ADR(ReadErr));
			pRxData := cl2.GetMessageDataPointer(hMessage:= hMsg,peError:=ADR(ReadErr));	
			Chassis_speed := pRxData^[7];
			cl2.FreeMessage(hMsg);
			nReceived := cl2.GetMsgCount(hReceiverId :=hReceiver_speed, peError := ADR(ReadErr));
		END_WHILE

		//接收底盘信息: ID:0x182126f4,  byte0*0.4  剩余SOC百分比
		nReceived := cl2.GetMsgCount(hReceiverId :=hReceiver_soc, peError := ADR(ReadErr));
		h:=h+1;
		WHILE nReceived > 0 DO
			h:=0;
			hMsg := cl2.Read(hReceiverId :=hReceiver_soc,pctMsgLeft:=ADR(nAvailable),peError:=ADR(ReadErr));
			pRxData := cl2.GetMessageDataPointer(hMessage:= hMsg,peError:=ADR(ReadErr));	
			tmp_uint := ANY_TO_UINT(pRxData^[0]);
			Chassis_Soc := ANY_TO_BYTE(tmp_uint*2/5);
			cl2.FreeMessage(hMsg);
			nReceived := cl2.GetMsgCount(hReceiverId :=hReceiver_soc, peError := ADR(ReadErr));		
		END_WHILE
	
         //电机驱动器CAN通讯判断
		 T_Chassis_CAN_fault(IN:=h>200,PT:=T#1S);
		 
			//底盘电量判断
		T_SOC_LOW(in:=(Chassis_Soc<20)AND NOT T_Chassis_CAN_fault.Q,PT:=T#2S);(*底盘电量低停机*)	
        Chassis_SOC_LOW:=T_SOC_LOW.Q;
//		IF Chassis_SOC_LOW THEN
//			a:=TRUE;
//		END_IF
		T_Chassis_SOC_LOW(in:=Chassis_SOC_LOW AND NOT T_Chassis_CAN_fault.Q,PT:=T#8S);(*底盘电量低停机*)
		

		
		
		can_stat := 20;


	100:   //error
		
		
		
END_CASE

END_PROGRAM

// Changsha_Xiangji_ARM_Cortex_A9_xilinx_zynq7000_linux/Application/CAN_COMM/prg_test_can
PROGRAM prg_test_can
VAR
	hCan0:CAA.HANDLE:=0;
	hCan1:CAA.HANDLE:=0;
	cmd_test:BOOL := FALSE;
    CanWriteData : ARRAY[0..7] OF BYTE;
    CanWriteMsgID:UDINT;
	CanReadData : ARRAY[0..7] OF BYTE;  
	CanReadMsgID:UDINT;		
	test_01:BOOL := FALSE;
	test_02:BOOL := FALSE;
	test_03:BOOL := FALSE;
	test_04:BOOL := FALSE;
	test_05:BOOL := FALSE;
	test_06:BOOL := FALSE;
	test_07:BOOL := FALSE;
	
END_VAR


IF NOT cmd_test THEN 
	RETURN;
END_IF

hCan0 := prg_can0.hCan0;
hCan1 := prg_can1.hCan1;

IF test_01 THEN
	CanWriteData[0] := 123;
	CanWriteData[1] := 1;
	CanWriteData[6] := 234;
	CAN_Send_MSG(hCan0, 16#0C112AEE, 8, CanWriteData);	
	test_01 := FALSE;
END_IF

IF test_02 THEN
	CAN_Send_MSG(hCan0, 16#0C122AEE, 8, CanWriteData);	
	test_02 := FALSE;
END_IF

IF test_03 THEN
	CAN_Send_MSG(hCan0, 16#0C132AEE, 8, CanWriteData);
	test_03 := FALSE;	
END_IF

IF test_04 THEN
	CAN_Send_MSG(hCan1, 16#18C21726, 8, CanWriteData);
	test_04 := FALSE;	
END_IF

END_PROGRAM

// Changsha_Xiangji_ARM_Cortex_A9_xilinx_zynq7000_linux/Application/GPRS/prg_gprs
PROGRAM prg_gprs
VAR
	is_inited :BOOL := FALSE;
	
	udp_handle :CAA.HANDLE; 
	udp_init_fb:Udp_Init;
	udp_write_fb:Udp_Write;
	udp_read_fb:Udp_Read;
	file_read_fb:File_Read;
	com_read_fb :Com_Read;
	packet_heart_fb:Packet_Heart;

	size :CAA.SIZE;	
	Writebuffer: 			ARRAY[1..200] OF BYTE;
	Readbuffer: 			ARRAY[0..1499] OF BYTE;
	ReadbufferStr: STRING;
	atcState :INT := 0;
	
	writeUdpState :INT := 0;
	readUdpState :INT := 0;
	
	i :INT;
	count :INT := 0;
	
	rtc_fb: RTC;
	dtu_set_dt_fb: dtu.SetDateAndTime;
	
	sn_file_name :STRING := '/userapp/sn.txt';
	time_file_name :STRING := '/userapp/r_mins.txt';
	is_read :BOOL := FALSE;
	read_count :INT := 0;
	readFileState :INT := 0;
	ton_fb :TON;
	accid_cmd :STRING := 'AT+ICCID$r';
	iccid_read_buffer :STRING;
	position :INT := -1;
	new_date:DT;
END_VAR

CASE readFileState OF
	0:
		file_read_fb(file_name := sn_file_name);
		is_read := file_read_fb.isRead;
		IF is_read THEN
			GVL.sn := file_read_fb.sReadLine;
			readFileState := 1;
		END_IF
	
	1:
		file_read_fb(file_name := time_file_name);
		is_read := file_read_fb.isRead;
		IF is_read THEN
			GVL.work_time := STRING_TO_UDINT(file_read_fb.sReadLine);
			readFileState := 2;
		END_IF
	
	2:
END_CASE


IF NOT is_inited THEN
	udp_init_fb(ip_addr := '47.107.240.29', port := 34567);
	IF udp_init_fb.init_mode = 1 THEN
		is_inited := TRUE;
		udp_handle := udp_init_fb.udp_handle;
		atcState := 2;
		Writebuffer[1] := 16#00;
		Writebuffer[2] := 16#01;
		Writebuffer[3] := 16#00;
		Writebuffer[4] := 16#01;
		Writebuffer[5] := 16#00;
		Writebuffer[6] := 16#14;
		Writebuffer[7] := 16#00;
		Writebuffer[8] := 16#00;
		Writebuffer[9] := 16#00;
		Writebuffer[10] := 16#04;
		Writebuffer[11] := 16#00;
		Writebuffer[12] := 16#00;
		Writebuffer[13] := 16#01;
		Writebuffer[14] := 16#88;
		Writebuffer[15] := 16#12;
		Writebuffer[16] := 16#34;
		Writebuffer[17] := 16#56;
		Writebuffer[18] := 16#78;
		Writebuffer[19] := 16#00;
		Writebuffer[20] := 16#01;
		Writebuffer[21] := 16#90;
	END_IF
END_IF


IF is_inited = TRUE THEN
	CASE atcState OF
	0:
	GVL.lac := 0;
	GVL.cid := 0;
	GVL.iccid := '';	
	com_read_fb(com:= udp_handle, wbuffer:= ADR(accid_cmd), wsize := len(accid_cmd), rbuffer := ADR(iccid_read_buffer), rsize := SIZEOF(iccid_read_buffer));
	IF com_read_fb.atcState = 255 THEN
		size := com_read_fb.size;
		atcState := 1;	
		IF size > 0 THEN
			position := find(iccid_read_buffer, '+ICCID:');
			IF position > 0 THEN
				GVL.iccid := mid(iccid_read_buffer, 20, position + len('+ICCID:'));
				atcState := 1;
			END_IF
		END_IF
	ELSIF com_read_fb.atcState = 32767 THEN
		atcState := 1;
	END_IF
	
	1:
	udp_write_fb(com := udp_handle, buffer:= ADR(Writebuffer), size := 21);
	writeUdpState := udp_write_fb.atcState;
	IF writeUdpState = 255 THEN
		atcState := 2;
	END_IF
		
	2:
	ton_fb(IN := TRUE, PT := TIME#500MS);
	IF (ton_fb.Q) THEN
		ton_fb(IN := FALSE, PT := TIME#500MS);
		atcState := 3;
	END_IF	
		
	3:
	udp_read_fb(com:= udp_handle, buffer:= ADR(Readbuffer), rsize := SIZEOF(Readbuffer));
	readUdpState := udp_read_fb.atcState;
	
	IF readUdpState = 32767 THEN
		atcState := 1;
	ELSIF readUdpState = 255 THEN
		atcState := 1;
		size := udp_read_fb.size;
		IF size > 0 THEN
			atcState := 4;
			FOR i := 0 TO 18 DO
				ReadbufferStr[0 + i] := Readbuffer[20 + i];  //21-->20
			END_FOR;
			
			ReadbufferStr[10] := 16#2D;
			ReadbufferStr[19] := 0;
			//rtc_fb(EN:=TRUE, PDT:=STRING_TO_DT(ReadbufferStr));
			new_date := STRING_TO_DT(ReadbufferStr);
			dtu_set_dt_fb.dtDateAndTime := new_date;
			dtu_set_dt_fb.xExecute := TRUE;
		END_IF
	END_IF
		
	4:
	IF dtu_set_dt_fb.xDone OR dtu_set_dt_fb.xError THEN
		dtu_set_dt_fb(xExecute := FALSE);	
	END_IF
	IF readFileState = 2 THEN
		packet_heart_fb(device_sn := GVL.sn, iccd_str := GVL.iccid, lac_num := GVL.lac, cid_num := GVL.cid, worktime := GVL.work_time);
		udp_write_fb(com := udp_handle, buffer:= ADR(packet_heart_fb.heart_buffer), size := 95);//size代表传送多少BYTE
		writeUdpState := udp_write_fb.atcState;
		IF writeUdpState = 255 THEN
			atcState := 5;
		END_IF
	END_IF
		
	5:	
	IF dtu_set_dt_fb.xDone OR dtu_set_dt_fb.xError THEN
		dtu_set_dt_fb(xExecute := FALSE);	
	END_IF	
	ton_fb(IN := TRUE, PT := TIME#10S);
	IF (ton_fb.Q) THEN
		ton_fb(IN := FALSE, PT := TIME#10S);
		atcState := 4;
	END_IF
		
	32767:
	
	END_CASE	
END_IF

dtu_set_dt_fb();

END_PROGRAM

// Changsha_Xiangji_ARM_Cortex_A9_xilinx_zynq7000_linux/Application/GPRS/File_Read
FUNCTION_BLOCK File_Read
VAR_INPUT
	file_name :STRING;
END_VAR
VAR_OUTPUT
	sReadLine		: STRING;
	isRead          :BOOL := FALSE;	
END_VAR
VAR
	hfile			: CAA.HANDLE;
	FileOpen 		: File.Open;
	FileClose		: File.Close;
	FileRead		: File.Read;
	
	iState			: UINT := 0;	
	xError			: BOOL := FALSE;
END_VAR

 CASE iState OF
	0: // Open the file again, with read access.
	   isRead := false;
	   FileOpen(xExecute:= TRUE, sFileName:= file_name, xExclusive:= FALSE, eFileMode:= File.MODE.MREAD);
	   IF FileOpen.xDone = TRUE THEN
		   hfile := FileOpen.hFile;
		   FileOpen(xExecute:= FALSE);
		   iState := 1;
		   sReadLine := '';
	   ELSIF FileOpen.xError = TRUE THEN
		   iState:= 32767;
		   FileOpen(xExecute:= FALSE);
	   END_IF

	1: // Read the string from the file.
	   FileRead(xExecute:= TRUE, hFile:= hfile, pBuffer:= ADR(sReadLine), szBuffer:= SIZEOF(sReadLine));
	   IF FileRead.xDone = TRUE THEN
		   iState := 2;		   
		   sReadLine := MID(sReadLine, ANY_TO_INT(FileRead.szSize), 1);
		   FileRead(xExecute:= FALSE);
	   ELSIF FileRead.xError = TRUE THEN
		   iState:= 32767;
		   FileRead(xExecute:= FALSE);
	   END_IF 
	   
	 2: // Close that file.
	   FileClose(xExecute:= TRUE, hFile:= hfile);
	   IF FileClose.xDone = TRUE THEN
		   iState := 3;
		   FileClose(xExecute:= FALSE);
	   ELSIF FileClose.xError = TRUE THEN
		   iState:= 32767;
		   FileClose(xExecute:= FALSE);
	   END_IF
	   
	3: 	  
		isRead := TRUE;
		iState := 0;
		
	32767: 		
	
END_CASE

END_FUNCTION_BLOCK

// Changsha_Xiangji_ARM_Cortex_A9_xilinx_zynq7000_linux/Application/GPRS/Packet_Heart
FUNCTION_BLOCK Packet_Heart
VAR_INPUT
	device_sn :STRING;
	iccd_str :STRING;
	lac_num :UINT;
	cid_num :UINT;
	worktime :UDINT;
END_VAR
VAR_OUTPUT
	heart_buffer : ARRAY[0..250] OF BYTE;
END_VAR
VAR
	heart_state :INT := 0;
	sub_str :STRING;
	num :UINT;
	packet_seq :BYTE := 0;
	iccid_code :ARRAY[0..9] OF BYTE;
	i : INT;
	
	total :UINT := 0;
	
END_VAR

//1. CMA123456781234
//1.1 CMA
heart_buffer[0] := device_sn[0];
heart_buffer[1] := device_sn[1];
heart_buffer[2] := device_sn[2];

// 1.2 12
sub_str := mid(device_sn, 2, 4);
heart_buffer[3] := STRING_TO_BYTE(sub_str);

// 1.3 34
sub_str := mid(device_sn, 2, 6);
heart_buffer[4] := STRING_TO_BYTE(sub_str);

// 1.4 56
sub_str := mid(device_sn, 2, 8);
heart_buffer[5] := STRING_TO_BYTE(sub_str);

// 1.5 78
sub_str := mid(device_sn, 2, 10);
heart_buffer[6] := STRING_TO_BYTE(sub_str);

// 1.6 1234
sub_str := mid(device_sn, 4, 12);
num := STRING_TO_UINT(sub_str);
heart_buffer[7] := ANY_TO_BYTE(num / 256);
heart_buffer[8] := ANY_TO_BYTE(num MOD 256);

// 2. protocol version
heart_buffer[9] := 0;

// 3. data length
heart_buffer[10] := 0;
heart_buffer[11] := 81;

// 4. data type
heart_buffer[12] := 16#01;

// 5. data seq
heart_buffer[13] := packet_seq;
packet_seq := packet_seq + 1;

// 6. parameter
heart_buffer[14] := 0;

// 7. version
heart_buffer[15] := 0;

// 8. reserved 1
heart_buffer[16] := 0;

// 9. reserved 2
heart_buffer[17] := 0;

// 10. length
heart_buffer[18] := 0;
heart_buffer[19] := 73;

// 11. LAC 
heart_buffer[20] := ANY_TO_BYTE(lac_num / 256);
heart_buffer[21] := ANY_TO_BYTE(lac_num MOD 256);

// 12. CID 
heart_buffer[22] := ANY_TO_BYTE(cid_num / 256);
heart_buffer[23] := ANY_TO_BYTE(cid_num MOD 256);

// 13. iccid
iccid_code := Iccid_Get(iccd_str);
FOR i := 0 TO 9 DO
	heart_buffer[24 + i] := iccid_code[i];
END_FOR

// 14. work time
heart_buffer[34] := ANY_TO_BYTE(worktime / 65536 /256);
heart_buffer[35] := ANY_TO_BYTE(worktime / 65536 MOD 256);
heart_buffer[36] := ANY_TO_BYTE(worktime MOD 65536 / 256);
heart_buffer[37] := ANY_TO_BYTE(worktime MOD 65536 MOD 256);

// 15. customer code
heart_buffer[38] := 0;
heart_buffer[39] := 0;

// 16. local host code
heart_buffer[40] := 0;
heart_buffer[41] := 0;

//**********以下为GPRS回传数据**************//
heart_buffer[42].0 := FALSE;
heart_buffer[42].1 := FALSE;
heart_buffer[42].2 := FALSE;
heart_buffer[42].3 := FALSE;
heart_buffer[42].4 := FALSE;
heart_buffer[42].5 := FALSE;
heart_buffer[42].6 := FALSE;
heart_buffer[42].7 := FALSE;

heart_buffer[43].0 := FALSE;
heart_buffer[43].1 := Wastewater_full_Fault;//污水满故障
heart_buffer[43].2 := T_DI_oil_filter_block.Q;//回油过滤堵塞
heart_buffer[43].3 := T_DI_oil_level_low.Q;//液压油位低故障
heart_buffer[43].4 := FALSE;
heart_buffer[43].5 := T_DI_cleanwater_LOW.Q;//水箱缺水故障
heart_buffer[43].6 := FALSE;
heart_buffer[43].7 := DI_Rcar_fault;//倒车故障停机

heart_buffer[44].0 := Wastewater_full_Fault1;//污水满故障停机
heart_buffer[44].1 := NOT DI_power_on;//电源故障
heart_buffer[44].2 := T_Pumpspeed_H.Q;//高压水泵超速报警
heart_buffer[44].3 := T_Pumpspeed_HH.Q;//高压水泵超速停止
heart_buffer[44].4 := TEST_ALM;//请关闭测试
heart_buffer[44].5 := RCAR_ALM;//正在倒车中提示
heart_buffer[44].6 := Motor_Work_ALM;//请先启动电机提示
heart_buffer[44].7 := Func_test_HMI;//测试打开

heart_buffer[45].0 := T_DI_air_press_low.Q;//气路系统压力低
heart_buffer[45].1 := T_DI_Rcar.Q;//倒车
heart_buffer[45].2 := FALSE;
heart_buffer[45].3 := DO_Hpre_pump_noWork;//高压水泵未啮合
heart_buffer[45].4 := T_Chassis_SOC_LOW.Q;//底盘电量低停机
heart_buffer[45].5 := DI_Hpre_valve_noOpen;//高压吹净球阀未打开
heart_buffer[45].6 := DI_Totvalve_noOpen;//高压水路球阀未打开
heart_buffer[45].7 := DO_Box_Up_arm;//请先打开箱门

heart_buffer[46].0 := fog_Spump_arm;//隔膜泵球阀未打开
heart_buffer[46].1 := T_fog_pump_press_noOk.Q;//隔膜泵压力不正常
heart_buffer[46].2 := Fault_STOP;//故障停机
heart_buffer[46].3 := DO_Box_Down_arm;//请先放下撑杆
heart_buffer[46].4 := T_DI_wastewater_full.Q;//主污水箱水满
heart_buffer[46].5 := Backup_power_Test_warn;//请先打开备用动力开关
heart_buffer[46].6 := T_Chassis_CAN_fault.Q;//底盘CAN通讯故障
heart_buffer[46].7 := T_Motor_CAN_fault.Q;//与电机CAN通讯故障

heart_buffer[47].0 := T_auxiliary_warte_dif.Q;//辅污水箱水位不一致
heart_buffer[47].1 := T_DI_auxiliary1_warte_H.Q;//辅1污水箱水满
heart_buffer[47].2 := T_DI_auxiliary2_warte_H.Q;//辅2污水箱水满
heart_buffer[47].3 := T_water_overflow_noClose.Q;//水路卸荷阀未关闭故障
heart_buffer[47].4 := T_water_overflow_noOpen.Q;//水路卸荷阀未打开故障
heart_buffer[47].5 := DI_backup_power_open;//备用动力打开提示
heart_buffer[47].6 := Chassis_SOC_LOW;//底盘电量低压20%提示
heart_buffer[47].7 := High_voltage_noReady;//底盘未上高压提示

heart_buffer[48].0 := (DI_cleanwater_LOW<3000);
heart_buffer[48].1 := DI_Totvalve_Open;
heart_buffer[48].2 := DI_box_door_close;
heart_buffer[48].3 := DI_Hpre_valve_open;
heart_buffer[48].4 := DI_air_press_low;
heart_buffer[48].5 := DI_wastewater_full;
heart_buffer[48].6 := DI_Rod_noDown;
heart_buffer[48].7 := DI_backup_power_open;

heart_buffer[49].0 := DI_water_overflow;
heart_buffer[49].1 := FALSE;
heart_buffer[49].2 := FALSE;
heart_buffer[49].3 := FALSE;
heart_buffer[49].4 := DI_fog_pump_press_ok;
heart_buffer[49].5 := DI_oil_level_low;
heart_buffer[49].6 := DI_oil_filter_block;
heart_buffer[49].7 := FALSE;

heart_buffer[50].0 := DI_power_on;
heart_buffer[50].1 := DI_Rcar;
heart_buffer[50].2 := DI_oil_release_valve;
heart_buffer[50].3 := FALSE;
heart_buffer[50].4 := DI_auxiliary1_warte_H;
heart_buffer[50].5 := DI_auxiliary2_warte_H;
heart_buffer[50].6 := DI_Sweep_Up;
heart_buffer[50].7 := DI_Sweep_Down;

heart_buffer[51].0 := DI_sweep_out;
heart_buffer[51].1 := DI_sweep_return;
heart_buffer[51].2 := FALSE;
heart_buffer[51].3 := FALSE;
heart_buffer[51].4 := FALSE;
heart_buffer[51].5 := FALSE;
heart_buffer[51].6 := FALSE;
heart_buffer[51].7 := FALSE;

heart_buffer[52].0 := DO_Lsweep_down;
heart_buffer[52].1 := DO_Lsweep_up;
heart_buffer[52].2 := DO_Rsweep_down;
heart_buffer[52].3 := DO_Rsweep_up;
heart_buffer[52].4 := DO_Lsweep_out;
heart_buffer[52].5 := DO_Rsweep_out;
heart_buffer[52].6 := DO_Lrod_out;
heart_buffer[52].7 := DO_Rrod_out;

heart_buffer[53].0 := DO_pointshoot_up;
heart_buffer[53].1 := DO_pointshoot_down;
heart_buffer[53].2 := DO_pointshoot_left;
heart_buffer[53].3 := DO_pointshoot_right;
heart_buffer[53].4 := FALSE;
heart_buffer[53].5 := DO_water_overflow;
heart_buffer[53].6 := DO_Lrod_water;
heart_buffer[53].7 := DO_Rrod_water;

heart_buffer[54].0 := DO_Suction_water;
heart_buffer[54].1 := DO_Hpressure_water;
heart_buffer[54].2 := DO_selfclean_water;
heart_buffer[54].3 := DO_Hpre_pump;
heart_buffer[54].4 := DO_fog_Spump;
heart_buffer[54].5 := DO_Motor_en;
heart_buffer[54].6 := DO_watercooler_pump;
heart_buffer[54].7 := DO_cooler_fan;

heart_buffer[55].0 := DO_backup_power;
heart_buffer[55].1 := DO_wastewater_valve;
heart_buffer[55].2 := DO_wastewater_pump;
heart_buffer[55].3 := DO_oil_release_valve;
heart_buffer[55].4 := DO_Sweep_Mspeed;
heart_buffer[55].5 := DO_Sweep_Lspeed;
heart_buffer[55].6 := DO_RSweep;
heart_buffer[55].7 := DO_LASweep;

heart_buffer[56].0 := DO_RASweep;
heart_buffer[56].1 := DO_Box_Down;
heart_buffer[56].2 := DO_Box_Up;
heart_buffer[56].3 := DO_Suction_Down;
heart_buffer[56].4 := DO_Suction_Up;
heart_buffer[56].5 := DO_Door_Open;
heart_buffer[56].6 := DO_Door_Close;
heart_buffer[56].7 := FALSE;

heart_buffer[57].0 := FALSE;
heart_buffer[57].1 := FALSE;
heart_buffer[57].2 := FALSE;
heart_buffer[57].3 := FALSE;
heart_buffer[57].4 := FALSE;
heart_buffer[57].5 := FALSE;
heart_buffer[57].6 := FALSE;
heart_buffer[57].7 := FALSE;

heart_buffer[58].0 := AwashSweep_HMI;
heart_buffer[58].1 := LwashSweep_HMI;
heart_buffer[58].2 := RwashSweep_HMI;
heart_buffer[58].3 := ASweeproad_HMI;
heart_buffer[58].4 := LSweeproad_HMI;
heart_buffer[58].5 := RSweeproad_HMI;
heart_buffer[58].6 := Aclean_HMI;
heart_buffer[58].7 := Lclean_HMI;

heart_buffer[59].0 := Rclean_HMI;
heart_buffer[59].1 := Sweep_stop_HMI;
heart_buffer[59].2 := DO_fog_Spump1;
heart_buffer[59].3 := DO_selfclean_water1;
heart_buffer[59].4 := DO_Door_Close1;
heart_buffer[59].5 := DO_Door_Open1;
heart_buffer[59].6 := DO_Box_Up1;
heart_buffer[59].7 := DO_Box_Down1;

heart_buffer[60].0 := FALSE;
heart_buffer[60].1 := FALSE;
heart_buffer[60].2 := FALSE;
heart_buffer[60].3 := FALSE;
heart_buffer[60].4 := Standard_speed_HMI;
heart_buffer[60].5 := Strong_speed_HMI;
heart_buffer[60].6 := Sweep_HSpeed_HMI;
heart_buffer[60].7 := Sweep_MSpeed_HMI;

heart_buffer[61].0 := Sweep_LSpeed_HMI;
heart_buffer[61].1 := DO_Hpressure_water1;
heart_buffer[61].2 := Drain_start_HMI;
heart_buffer[61].3 := Drain_auto_HMI;
heart_buffer[61].4 := Drain_manual_HMI;
heart_buffer[61].5 := Lrod_drain_HMI;
heart_buffer[61].6 := Rrod_drain_HMI;
heart_buffer[61].7 := Hpressure_drain_HMI;

heart_buffer[62].0 := Selfclean_drain_HMI;
heart_buffer[62].1 := replace_Sweep_HMI;
heart_buffer[62].2 := Func_test_HMI;
heart_buffer[62].3 := Intelligent_HMI;
heart_buffer[62].4 := Cleanly_HMI;
heart_buffer[62].5 := Normal_HMI;
heart_buffer[62].6 := Dirty_HMI;
heart_buffer[62].7 := DO_wastewater_pump_open1;

heart_buffer[63].0 := Pointshoot_up_HMI;
heart_buffer[63].1 := Pointshoot_down_HMI;
heart_buffer[63].2 := Pointshoot_left_HMI;
heart_buffer[63].3 := Pointshoot_right_HMI;
heart_buffer[63].4 := Suction_drain_HMI;
heart_buffer[63].5 := FALSE;
heart_buffer[63].6 := motor_work;
heart_buffer[63].7 := sys_work;

heart_buffer[64] := ANY_TO_BYTE(Motor_real_torque_HMI MOD 256);
heart_buffer[65] :=ANY_TO_BYTE(Motor_real_torque_HMI/256);

heart_buffer[66] :=ANY_TO_BYTE(Motor_real_speed_HMI MOD 256);
heart_buffer[67] :=ANY_TO_BYTE(Motor_real_speed_HMI/256);

heart_buffer[68] :=ANY_TO_BYTE(Motor_bus_voltage_HMI MOD 256);
heart_buffer[69] :=ANY_TO_BYTE(Motor_bus_voltage_HMI/256);

heart_buffer[70] :=ANY_TO_BYTE(Motor_phase_current_HMI MOD 256);
heart_buffer[71] :=ANY_TO_BYTE(Motor_phase_current_HMI/256);

heart_buffer[72] :=ANY_TO_BYTE(Motor_max_dirve_torque_HMI MOD 256);
heart_buffer[73] :=ANY_TO_BYTE(Motor_max_dirve_torque_HMI/256);

heart_buffer[74] :=ANY_TO_BYTE(Motor_max_brake_torque_HMI MOD 256);
heart_buffer[75] :=ANY_TO_BYTE(Motor_max_brake_torque_HMI/256);

heart_buffer[76] :=Motor_temp_controller_HMI;
heart_buffer[77] :=Motor_temp_HMI;

heart_buffer[78] :=ANY_TO_BYTE(Motor_max_speed_HMI MOD 256);
heart_buffer[79] :=ANY_TO_BYTE(Motor_max_speed_HMI/256);

heart_buffer[80] := 0*1+Motor_direction_cw*4+Motor_mode*16+Motor_stat*64;
heart_buffer[81] := Motor_bus_low_voltage*1+Motor_bus_high_voltage*4+MOtor_ctrller_high_temp*16+Motor_high_temp*64;
heart_buffer[82] := Motor_igbt_fault*1+Motor_overspeed*4+Motor_comm_error*16+Motor_short*64;
heart_buffer[83] := Motor_overload*1+Motor_selfcheck_fault*4+Motor_low_voltage*16+Motor_sensor_fault*64;

heart_buffer[84] := Chassis_Soc;//底盘电量

heart_buffer[85] :=ANY_TO_BYTE(16#201 MOD 256);
heart_buffer[86] :=ANY_TO_BYTE(16#201/256);

heart_buffer[87] :=ANY_TO_BYTE(Chassis_speed MOD 256);
heart_buffer[88] :=ANY_TO_BYTE(Chassis_speed/256);//底盘车速

heart_buffer[89] :=ANY_TO_BYTE(motor_work_time MOD 256);
heart_buffer[90] :=ANY_TO_BYTE(motor_work_time/16#100);
heart_buffer[91] :=ANY_TO_BYTE(motor_work_time/16#10000);
heart_buffer[92] :=ANY_TO_BYTE(motor_work_time/16#1000000);


//**********以上为GPRS回传数据**************//

//以下为校验需要放到最后
total := 0;
FOR i := 0 TO 92 DO    (* 90代表GPRS回传的数据字节总数 *)
	total := total + heart_buffer[i];
END_FOR

// 15. taotal check
heart_buffer[93] := ANY_TO_BYTE(total / 256);
heart_buffer[94] := ANY_TO_BYTE(total MOD 256);

END_FUNCTION_BLOCK

// Changsha_Xiangji_ARM_Cortex_A9_xilinx_zynq7000_linux/Application/GPRS/Iccid_Get
FUNCTION Iccid_Get : ARRAY[0..9] OF BYTE
VAR_INPUT
	iccd :STRING;
END_VAR
VAR
	iccid_code :ARRAY[0..9] OF BYTE;
	
	byteHigh :BYTE := 0;
	byteLow :BYTE := 0;
	dstLen :INT := 0;
	
	srcIndex :INT := 0;
	bytesIndex :INT := 0;
END_VAR

dstLen := len(iccd) / 2;

FOR bytesIndex := 0 TO dstLen - 1 DO
	srcIndex := bytesIndex * 2;
	
	IF iccd[srcIndex] >= 16#30 AND iccd[srcIndex] <= 16#39 THEN
		byteHigh := iccd[srcIndex] - 16#30;
	ELSIF iccd[srcIndex] >= 16#41 AND iccd[srcIndex] <= 16#5A THEN
		byteHigh := iccd[srcIndex] - 55;
	END_IF
	
	IF iccd[srcIndex + 1] >= 16#30 AND iccd[srcIndex + 1] <= 16#39 THEN
		byteLow := iccd[srcIndex + 1] - 16#30;
	ELSIF iccd[srcIndex + 1] >= 16#41 AND iccd[srcIndex + 1] <= 16#5A THEN
		byteHigh := iccd[srcIndex + 1] - 55;
	END_IF
	
	iccid_code[bytesIndex] := byteHigh * 16 + byteLow;
END_FOR;

Iccid_Get := iccid_code;

END_FUNCTION

// Changsha_Xiangji_ARM_Cortex_A9_xilinx_zynq7000_linux/Application/main
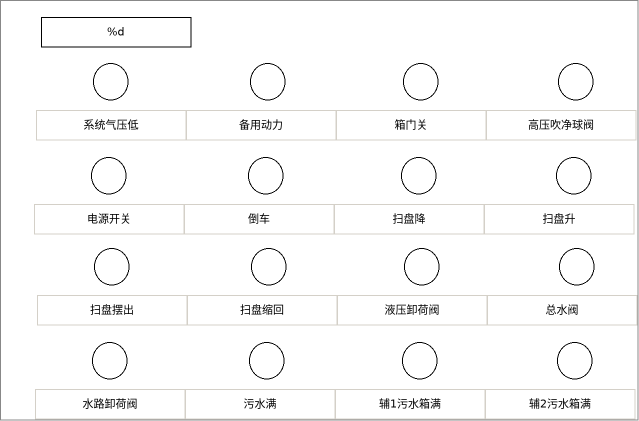
VISUALIZATION main  // 639x421
    RoundedRectangle (41,17 150x30), "%d", text variable: Motor_real_speed_HMI
    Ellipse (93,63 35x37), colour toggle: DI_air_press_low
    Textfield (36,110 150x30), "系统气压低"
    Ellipse (250,63 35x37), colour toggle: DI_backup_power_open
    Textfield (186,110 150x30), "备用动力"
    Ellipse (403,63 35x37), colour toggle: DI_box_door_close
    Textfield (336,110 150x30), "箱门关"
    Ellipse (558,63 35x37), colour toggle: DI_Hpre_valve_open
    Textfield (486,110 150x30), "高压吹净球阀"
    Ellipse (91,157 35x37), colour toggle: DI_power_on
    Textfield (34,204 150x30), "电源开关"
    Ellipse (248,157 35x37), colour toggle: DI_Rcar
    Textfield (184,204 150x30), "倒车"
    Ellipse (401,157 35x37), colour toggle: DI_Sweep_Down
    Textfield (334,204 150x30), "扫盘降"
    Ellipse (556,157 35x37), colour toggle: DI_Sweep_Up
    Textfield (484,204 150x30), "扫盘升"
    Ellipse (94,248 35x37), colour toggle: DI_sweep_out
    Textfield (37,295 150x30), "扫盘摆出"
    Ellipse (251,248 35x37), colour toggle: DI_sweep_return
    Textfield (187,295 150x30), "扫盘缩回"
    Ellipse (404,248 35x37), colour toggle: DI_oil_release_valve
    Textfield (337,295 150x30), "液压卸荷阀"
    Ellipse (559,248 35x37), colour toggle: DI_Totvalve_Open
    Textfield (487,295 150x30), "总水阀"
    Ellipse (92,342 35x37), colour toggle: DI_water_overflow
    Textfield (35,389 150x30), "水路卸荷阀"
    Ellipse (249,342 35x37), colour toggle: DI_wastewater_full
    Textfield (185,389 150x30), "污水满"
    Ellipse (402,342 35x37), colour toggle: DI_auxiliary1_warte_H
    Textfield (335,389 150x30), "辅1污水箱满"
    Ellipse (557,342 35x37), colour toggle: DI_auxiliary2_warte_H
    Textfield (485,389 150x30), "辅2污水箱满"
END_VISUALIZATION
